LIN {X 0,Y 474.103,Z 226.127,A -85,B 0,C 180,E1 22326.053,E2 22326.053} C_VEL
LIN {X 0,Y 474.112,Z 226.175,A -85,B 0,C 180,E1 22322.417,E2 22322.417} C_VEL
LIN {X 0,Y 474.109,Z 226.126,A -85,B 0,C 180,E1 22318.792,E2 22318.792} C_VEL
LIN {X 0,Y 474.1,Z 226.168,A -85,B 0,C 180,E1 22315.161,E2 22315.161} C_VEL
LIN {X 0,Y 474.084,Z 226.14,A -85,B 0,C 180,E1 22311.559,E2 22311.559} C_VEL
LIN {X 0,Y 474.099,Z 226.178,A -85,B 0,C 180,E1 22307.948,E2 22307.948} C_VEL
LIN {X 0,Y 474.117,Z 226.162,A -85,B 0,C 180,E1 22304.339,E2 22304.339} C_VEL
LIN {X 0,Y 474.116,Z 226.167,A -85,B 0,C 180,E1 22300.664,E2 22300.664} C_VEL
LIN {X 0,Y 474.086,Z 226.178,A -85,B 0,C 180,E1 22297.165,E2 22297.165} C_VEL
LIN {X 0,Y 474.083,Z 226.168,A -85,B 0,C 180,E1 22293.575,E2 22293.575} C_VEL
LIN {X 0,Y 474.134,Z 226.296,A -85,B 0,C 180,E1 22292.55,E2 22292.55} C_VEL
LIN {X 0,Y 475.326,Z 229.528,A -85,B 0,C 180,E1 22292.024,E2 22292.024} C_VEL
LIN {X 0,Y 476.699,Z 231.84,A -85,B 0,C 180,E1 22291.566,E2 22291.566} C_VEL
LIN {X 0,Y 481.647,Z 241.457,A -85,B 0,C 180,E1 22289.842,E2 22289.842} C_VEL
LIN {X 0,Y 489.624,Z 256.766,A -85,B 0,C 180,E1 22287.236,E2 22287.236} C_VEL
LIN {X 0,Y 500.094,Z 277.627,A -85,B 0,C 180,E1 22283.997,E2 22283.997} C_VEL
LIN {X 0,Y 511.483,Z 301.22,A -85,B 0,C 180,E1 22280.7,E2 22280.7} C_VEL
LIN {X 0,Y 519.807,Z 318.56,A -85,B 0,C 180,E1 22278.514,E2 22278.514} C_VEL
LIN {X 0,Y 522.352,Z 322.995,A -85,B 0,C 180,E1 22278.188,E2 22278.188} C_VEL
LIN {X 0,Y 524.642,Z 347.742,A -85,B 0,C 180,E1 22277.464,E2 22277.464} C_VEL
LIN {X 0,Y 513.943,Z 587.488,A -85,B 0,C 180,E1 22273.462,E2 22273.462} C_VEL
LIN {X 0,Y 509.832,Z 692.964,A -85,B 0,C 180,E1 22271.722,E2 22271.722} C_VEL
LIN {X 0,Y 508.032,Z 717.442,A -85,B 0,C 180,E1 22271.132,E2 22271.132} C_VEL
LIN {X 0,Y 505.864,Z 741.406,A -85,B 0,C 180,E1 22270.37,E2 22270.37} C_VEL
LIN {X 0,Y 503.324,Z 764.227,A -85,B 0,C 180,E1 22269.435,E2 22269.435} C_VEL
LIN {X 0,Y 500.285,Z 788.254,A -85,B 0,C 180,E1 22268.236,E2 22268.236} C_VEL
LIN {X 0,Y 497.424,Z 808.594,A -85,B 0,C 180,E1 22267.016,E2 22267.016} C_VEL
LIN {X 0,Y 493.885,Z 831.697,A -85,B 0,C 180,E1 22265.382,E2 22265.382} C_VEL
LIN {X 0,Y 490.913,Z 850.192,A -85,B 0,C 180,E1 22263.853,E2 22263.853} C_VEL
LIN {X 0,Y 487.599,Z 870.092,A -85,B 0,C 180,E1 22261.942,E2 22261.942} C_VEL
LIN {X 0,Y 484.649,Z 887.507,A -85,B 0,C 180,E1 22260.02,E2 22260.02} C_VEL
LIN {X 0,Y 481.773,Z 904.616,A -85,B 0,C 180,E1 22257.838,E2 22257.838} C_VEL
LIN {X 0,Y 479.426,Z 919.191,A -85,B 0,C 180,E1 22255.709,E2 22255.709} C_VEL
LIN {X 0,Y 477.164,Z 934.025,A -85,B 0,C 180,E1 22253.201,E2 22253.201} C_VEL
LIN {X 0,Y 475.501,Z 946.237,A -85,B 0,C 180,E1 22250.816,E2 22250.816} C_VEL
LIN {X 0,Y 474.103,Z 958.209,A -85,B 0,C 180,E1 22248.061,E2 22248.061} C_VEL
LIN {X 0,Y 473.22,Z 967.521,A -85,B 0,C 180,E1 22245.526,E2 22245.526} C_VEL
LIN {X 0,Y 472.64,Z 976.006,A -85,B 0,C 180,E1 22242.71,E2 22242.71} C_VEL
LIN {X 0,Y 472.385,Z 982.114,A -85,B 0,C 180,E1 22240.178,E2 22240.178} C_VEL
LIN {X 0,Y 472.289,Z 987.389,A -85,B 0,C 180,E1 22237.298,E2 22237.298} C_VEL
LIN {X 0,Y 472.333,Z 990.403,A -85,B 0,C 180,E1 22234.857,E2 22234.857} C_VEL
LIN {X 0,Y 472.382,Z 992.129,A -85,B 0,C 180,E1 22232.548,E2 22232.548} C_VEL
LIN {X 0,Y 472.425,Z 992.783,A -85,B 0,C 180,E1 22229.879,E2 22229.879} C_VEL
LIN {X 0,Y 472.4,Z 991.751,A -85,B 0,C 180,E1 22227.21,E2 22227.21} C_VEL
LIN {X 0,Y 472.366,Z 989.7,A -85,B 0,C 180,E1 22224.899,E2 22224.899} C_VEL
LIN {X 0,Y 472.343,Z 986.144,A -85,B 0,C 180,E1 22222.336,E2 22222.336} C_VEL
LIN {X 0,Y 472.457,Z 980.753,A -85,B 0,C 180,E1 22219.636,E2 22219.636} C_VEL
LIN {X 0,Y 472.711,Z 974.464,A -85,B 0,C 180,E1 22217.168,E2 22217.168} C_VEL
LIN {X 0,Y 473.282,Z 965.476,A -85,B 0,C 180,E1 22214.311,E2 22214.311} C_VEL
LIN {X 0,Y 474.142,Z 955.945,A -85,B 0,C 180,E1 22211.814,E2 22211.814} C_VEL
LIN {X 0,Y 475.522,Z 943.625,A -85,B 0,C 180,E1 22209.055,E2 22209.055} C_VEL
LIN {X 0,Y 477.241,Z 930.371,A -85,B 0,C 180,E1 22206.542,E2 22206.542} C_VEL
LIN {X 0,Y 479.545,Z 914.812,A -85,B 0,C 180,E1 22203.984,E2 22203.984} C_VEL
LIN {X 0,Y 482.006,Z 899.256,A -85,B 0,C 180,E1 22201.773,E2 22201.773} C_VEL
LIN {X 0,Y 485.194,Z 880.054,A -85,B 0,C 180,E1 22199.401,E2 22199.401} C_VEL
LIN {X 0,Y 488.36,Z 861.534,A -85,B 0,C 180,E1 22197.42,E2 22197.42} C_VEL
LIN {X 0,Y 491.865,Z 840.855,A -85,B 0,C 180,E1 22195.519,E2 22195.519} C_VEL
LIN {X 0,Y 495.389,Z 819.524,A -85,B 0,C 180,E1 22193.823,E2 22193.823} C_VEL
LIN {X 0,Y 498.74,Z 797.883,A -85,B 0,C 180,E1 22192.365,E2 22192.365} C_VEL
LIN {X 0,Y 502.253,Z 774.045,A -85,B 0,C 180,E1 22191.016,E2 22191.016} C_VEL
LIN {X 0,Y 505.228,Z 751.77,A -85,B 0,C 180,E1 22189.969,E2 22189.969} C_VEL
LIN {X 0,Y 507.919,Z 728.566,A -85,B 0,C 180,E1 22189.093,E2 22189.093} C_VEL
LIN {X 0,Y 510.279,Z 705.051,A -85,B 0,C 180,E1 22188.392,E2 22188.392} C_VEL
LIN {X 0,Y 512.094,Z 679.83,A -85,B 0,C 180,E1 22187.846,E2 22187.846} C_VEL
LIN {X 0,Y 517.017,Z 597.902,A -85,B 0,C 180,E1 22186.328,E2 22186.328} C_VEL
LIN {X 0,Y 522.642,Z 530.22,A -85,B 0,C 180,E1 22184.953,E2 22184.953} C_VEL
LIN {X 0,Y 529.867,Z 464.415,A -85,B 0,C 180,E1 22183.508,E2 22183.508} C_VEL
LIN {X 0,Y 538.765,Z 402.255,A -85,B 0,C 180,E1 22182.087,E2 22182.087} C_VEL
LIN {X 0,Y 544.168,Z 370.237,A -85,B 0,C 180,E1 22181.326,E2 22181.326} C_VEL
LIN {X 0,Y 538.418,Z 386.185,A -85,B 0,C 180,E1 22179.758,E2 22179.758} C_VEL
LIN {X 0,Y 534.921,Z 400.034,A -85,B 0,C 180,E1 22178.53,E2 22178.53} C_VEL
LIN {X 0,Y 531.61,Z 418.651,A -85,B 0,C 180,E1 22177.072,E2 22177.072} C_VEL
LIN {X 0,Y 528.747,Z 441.431,A -85,B 0,C 180,E1 22175.545,E2 22175.545} C_VEL
LIN {X 0,Y 526.309,Z 468.54,A -85,B 0,C 180,E1 22173.972,E2 22173.972} C_VEL
LIN {X 0,Y 524.021,Z 500.146,A -85,B 0,C 180,E1 22172.4,E2 22172.4} C_VEL
LIN {X 0,Y 523.085,Z 512.301,A -85,B 0,C 180,E1 22171.879,E2 22171.879} C_VEL
LIN {X 0,Y 507.968,Z 623.688,A -85,B 0,C 180,E1 22168.838,E2 22168.838} C_VEL
LIN {X 0,Y 500.211,Z 692.312,A -85,B 0,C 180,E1 22166.905,E2 22166.905} C_VEL
LIN {X 0,Y 497.222,Z 717.176,A -85,B 0,C 180,E1 22165.969,E2 22165.969} C_VEL
LIN {X 0,Y 494.515,Z 738.857,A -85,B 0,C 180,E1 22164.934,E2 22164.934} C_VEL
LIN {X 0,Y 491.751,Z 760.438,A -85,B 0,C 180,E1 22163.677,E2 22163.677} C_VEL
LIN {X 0,Y 489.036,Z 780.869,A -85,B 0,C 180,E1 22162.226,E2 22162.226} C_VEL
LIN {X 0,Y 486.605,Z 798.705,A -85,B 0,C 180,E1 22160.697,E2 22160.697} C_VEL
LIN {X 0,Y 484.482,Z 813.948,A -85,B 0,C 180,E1 22159.157,E2 22159.157} C_VEL
LIN {X 0,Y 482.34,Z 828.73,A -85,B 0,C 180,E1 22157.368,E2 22157.368} C_VEL
LIN {X 0,Y 480.502,Z 841.055,A -85,B 0,C 180,E1 22155.572,E2 22155.572} C_VEL
LIN {X 0,Y 478.852,Z 851.963,A -85,B 0,C 180,E1 22153.648,E2 22153.648} C_VEL
LIN {X 0,Y 477.393,Z 861.257,A -85,B 0,C 180,E1 22151.6,E2 22151.6} C_VEL
LIN {X 0,Y 476.233,Z 868.521,A -85,B 0,C 180,E1 22149.548,E2 22149.548} C_VEL
LIN {X 0,Y 475.29,Z 874.171,A -85,B 0,C 180,E1 22147.373,E2 22147.373} C_VEL
LIN {X 0,Y 474.594,Z 877.91,A -85,B 0,C 180,E1 22145.198,E2 22145.198} C_VEL
LIN {X 0,Y 474.097,Z 879.81,A -85,B 0,C 180,E1 22143.022,E2 22143.022} C_VEL
LIN {X 0,Y 473.788,Z 879.972,A -85,B 0,C 180,E1 22140.967,E2 22140.967} C_VEL
LIN {X 0,Y 473.605,Z 878.463,A -85,B 0,C 180,E1 22138.79,E2 22138.79} C_VEL
LIN {X 0,Y 473.549,Z 875.211,A -85,B 0,C 180,E1 22136.611,E2 22136.611} C_VEL
LIN {X 0,Y 473.645,Z 870.182,A -85,B 0,C 180,E1 22134.427,E2 22134.427} C_VEL
LIN {X 0,Y 473.915,Z 863.283,A -85,B 0,C 180,E1 22132.24,E2 22132.24} C_VEL
LIN {X 0,Y 474.405,Z 854.34,A -85,B 0,C 180,E1 22130.048,E2 22130.048} C_VEL
LIN {X 0,Y 475.124,Z 843.798,A -85,B 0,C 180,E1 22127.975,E2 22127.975} C_VEL
LIN {X 0,Y 476.057,Z 831.7,A -85,B 0,C 180,E1 22126.017,E2 22126.017} C_VEL
LIN {X 0,Y 477.184,Z 818.188,A -85,B 0,C 180,E1 22124.193,E2 22124.193} C_VEL
LIN {X 0,Y 478.539,Z 802.58,A -85,B 0,C 180,E1 22122.426,E2 22122.426} C_VEL
LIN {X 0,Y 480.003,Z 785.869,A -85,B 0,C 180,E1 22120.847,E2 22120.847} C_VEL
LIN {X 0,Y 481.552,Z 767.326,A -85,B 0,C 180,E1 22119.393,E2 22119.393} C_VEL
LIN {X 0,Y 483.066,Z 748.687,A -85,B 0,C 180,E1 22118.189,E2 22118.189} C_VEL
LIN {X 0,Y 484.603,Z 728.049,A -85,B 0,C 180,E1 22117.112,E2 22117.112} C_VEL
LIN {X 0,Y 486.002,Z 706.513,A -85,B 0,C 180,E1 22116.236,E2 22116.236} C_VEL
LIN {X 0,Y 487.201,Z 684.993,A -85,B 0,C 180,E1 22115.593,E2 22115.593} C_VEL
LIN {X 0,Y 491.38,Z 580.934,A -85,B 0,C 180,E1 22113.516,E2 22113.516} C_VEL
LIN {X 0,Y 494.767,Z 499.908,A -85,B 0,C 180,E1 22111.921,E2 22111.921} C_VEL
LIN {X 0,Y 489.856,Z 444.398,A -85,B 0,C 180,E1 22110.331,E2 22110.331} C_VEL
LIN {X 0,Y 494.577,Z 391.935,A -85,B 0,C 180,E1 22106.403,E2 22106.403} C_VEL
LIN {X 0,Y 499.626,Z 341.605,A -85,B 0,C 180,E1 22102.609,E2 22102.609} C_VEL
LIN {X 0,Y 504.089,Z 300.496,A -85,B 0,C 180,E1 22099.482,E2 22099.482} C_VEL
LIN {X 0,Y 497.077,Z 281.186,A -85,B 0,C 180,E1 22097.164,E2 22097.164} C_VEL
LIN {X 0,Y 498.864,Z 281.752,A -85,B 0,C 180,E1 22096.884,E2 22096.884} C_VEL
LIN {X 0,Y 503.777,Z 281.964,A -85,B 0,C 180,E1 22096.235,E2 22096.235} C_VEL
LIN {X 0,Y 511.406,Z 300.357,A -85,B 0,C 180,E1 22093.905,E2 22093.905} C_VEL
LIN {X 0,Y 517.83,Z 317.866,A -85,B 0,C 180,E1 22091.832,E2 22091.832} C_VEL
LIN {X 0,Y 517.363,Z 358.606,A -85,B 0,C 180,E1 22089.03,E2 22089.03} C_VEL
LIN {X 0,Y 513.648,Z 376.214,A -85,B 0,C 180,E1 22088.372,E2 22088.372} C_VEL
LIN {X 0,Y 510.519,Z 461.786,A -85,B 0,C 180,E1 22087.05,E2 22087.05} C_VEL
LIN {X 0,Y 507.289,Z 524.733,A -85,B 0,C 180,E1 22085.908,E2 22085.908} C_VEL
LIN {X 0,Y 506.039,Z 532.367,A -85,B 0,C 180,E1 22085.83,E2 22085.83} C_VEL
LIN {X 0,Y 499.793,Z 552.676,A -85,B 0,C 180,E1 22085.852,E2 22085.852} C_VEL
LIN {X 0,Y 498.777,Z 559.214,A -85,B 0,C 180,E1 22085.766,E2 22085.766} C_VEL
LIN {X 0,Y 493.831,Z 632.998,A -85,B 0,C 180,E1 22084.1,E2 22084.1} C_VEL
LIN {X 0,Y 492.338,Z 660.657,A -85,B 0,C 180,E1 22083.328,E2 22083.328} C_VEL
LIN {X 0,Y 490.752,Z 682.372,A -85,B 0,C 180,E1 22082.506,E2 22082.506} C_VEL
LIN {X 0,Y 488.846,Z 702.844,A -85,B 0,C 180,E1 22081.519,E2 22081.519} C_VEL
LIN {X 0,Y 486.522,Z 723.263,A -85,B 0,C 180,E1 22080.301,E2 22080.301} C_VEL
LIN {X 0,Y 483.983,Z 742.53,A -85,B 0,C 180,E1 22078.91,E2 22078.91} C_VEL
LIN {X 0,Y 481.322,Z 760.902,A -85,B 0,C 180,E1 22077.329,E2 22077.329} C_VEL
LIN {X 0,Y 478.596,Z 778.314,A -85,B 0,C 180,E1 22075.558,E2 22075.558} C_VEL
LIN {X 0,Y 476.006,Z 794.203,A -85,B 0,C 180,E1 22073.654,E2 22073.654} C_VEL
LIN {X 0,Y 473.532,Z 809.093,A -85,B 0,C 180,E1 22071.556,E2 22071.556} C_VEL
LIN {X 0,Y 471.329,Z 822.494,A -85,B 0,C 180,E1 22069.326,E2 22069.326} C_VEL
LIN {X 0,Y 469.449,Z 834.427,A -85,B 0,C 180,E1 22066.966,E2 22066.966} C_VEL
LIN {X 0,Y 467.909,Z 844.825,A -85,B 0,C 180,E1 22064.479,E2 22064.479} C_VEL
LIN {X 0,Y 466.793,Z 853.257,A -85,B 0,C 180,E1 22061.992,E2 22061.992} C_VEL
LIN {X 0,Y 466.006,Z 859.958,A -85,B 0,C 180,E1 22059.51,E2 22059.51} C_VEL
LIN {X 0,Y 465.509,Z 865.261,A -85,B 0,C 180,E1 22056.909,E2 22056.909} C_VEL
LIN {X 0,Y 465.23,Z 868.891,A -85,B 0,C 180,E1 22054.314,E2 22054.314} C_VEL
LIN {X 0,Y 465.099,Z 870.797,A -85,B 0,C 180,E1 22051.725,E2 22051.725} C_VEL
LIN {X 0,Y 465.069,Z 871.098,A -85,B 0,C 180,E1 22049.261,E2 22049.261} C_VEL
LIN {X 0,Y 465.149,Z 869.976,A -85,B 0,C 180,E1 22046.796,E2 22046.796} C_VEL
LIN {X 0,Y 465.356,Z 867.167,A -85,B 0,C 180,E1 22044.204,E2 22044.204} C_VEL
LIN {X 0,Y 465.713,Z 862.893,A -85,B 0,C 180,E1 22041.729,E2 22041.729} C_VEL
LIN {X 0,Y 466.373,Z 856.661,A -85,B 0,C 180,E1 22039.096,E2 22039.096} C_VEL
LIN {X 0,Y 467.313,Z 849.17,A -85,B 0,C 180,E1 22036.639,E2 22036.639} C_VEL
LIN {X 0,Y 468.657,Z 839.774,A -85,B 0,C 180,E1 22034.152,E2 22034.152} C_VEL
LIN {X 0,Y 470.425,Z 828.283,A -85,B 0,C 180,E1 22031.665,E2 22031.665} C_VEL
LIN {X 0,Y 472.548,Z 815.17,A -85,B 0,C 180,E1 22029.307,E2 22029.307} C_VEL
LIN {X 0,Y 474.847,Z 801.303,A -85,B 0,C 180,E1 22027.204,E2 22027.204} C_VEL
LIN {X 0,Y 477.37,Z 786.058,A -85,B 0,C 180,E1 22025.234,E2 22025.234} C_VEL
LIN {X 0,Y 480.042,Z 769.347,A -85,B 0,C 180,E1 22023.396,E2 22023.396} C_VEL
LIN {X 0,Y 482.71,Z 751.732,A -85,B 0,C 180,E1 22021.75,E2 22021.75} C_VEL
LIN {X 0,Y 485.282,Z 733.327,A -85,B 0,C 180,E1 22020.295,E2 22020.295} C_VEL
LIN {X 0,Y 487.727,Z 713.336,A -85,B 0,C 180,E1 22018.976,E2 22018.976} C_VEL
LIN {X 0,Y 489.988,Z 691.73,A -85,B 0,C 180,E1 22017.818,E2 22017.818} C_VEL
LIN {X 0,Y 491.801,Z 669.836,A -85,B 0,C 180,E1 22016.893,E2 22016.893} C_VEL
LIN {X 0,Y 493.107,Z 647.709,A -85,B 0,C 180,E1 22016.184,E2 22016.184} C_VEL
LIN {X 0,Y 495.899,Z 602.371,A -85,B 0,C 180,E1 22015.079,E2 22015.079} C_VEL
LIN {X 0,Y 500.552,Z 531.774,A -85,B 0,C 180,E1 22013.579,E2 22013.579} C_VEL
LIN {X 0,Y 504.112,Z 465.945,A -85,B 0,C 180,E1 22012.361,E2 22012.361} C_VEL
LIN {X 0,Y 507.201,Z 385.644,A -85,B 0,C 180,E1 22011.099,E2 22011.099} C_VEL
LIN {X 0,Y 507.596,Z 377.376,A -85,B 0,C 180,E1 22010.96,E2 22010.96} C_VEL
LIN {X 0,Y 511.408,Z 359.689,A -85,B 0,C 180,E1 22010.257,E2 22010.257} C_VEL
LIN {X 0,Y 511.798,Z 321.583,A -85,B 0,C 180,E1 22007.622,E2 22007.622} C_VEL
LIN {X 0,Y 503.702,Z 299.721,A -85,B 0,C 180,E1 22004.967,E2 22004.967} C_VEL
LIN {X 0,Y 495.259,Z 280.206,A -85,B 0,C 180,E1 22002.402,E2 22002.402} C_VEL
LIN {X 0,Y 487.022,Z 263.522,A -85,B 0,C 180,E1 21999.987,E2 21999.987} C_VEL
LIN {X 0,Y 480.126,Z 251.024,A -85,B 0,C 180,E1 21998.057,E2 21998.057} C_VEL
LIN {X 0,Y 474.875,Z 242.046,A -85,B 0,C 180,E1 21996.576,E2 21996.576} C_VEL
LIN {X 0,Y 472.072,Z 237.344,A -85,B 0,C 180,E1 21995.774,E2 21995.774} C_VEL
LIN {X 0,Y 469.994,Z 234.244,A -85,B 0,C 180,E1 21995.208,E2 21995.208} C_VEL
LIN {X 0,Y 469.308,Z 232.581,A -85,B 0,C 180,E1 21994.968,E2 21994.968} C_VEL
LIN {X 0,Y 467.108,Z 230.042,A -85,B 0,C 180,E1 21994.411,E2 21994.411} C_VEL
LIN {X 0,Y 466.171,Z 227.144,A -85,B 0,C 180,E1 21994.006,E2 21994.006} C_VEL
LIN {X 0,Y 466.183,Z 227.157,A -85,B 0,C 180,E1 21990.268,E2 21990.268} C_VEL
LIN {X 0,Y 466.167,Z 227.157,A -85,B 0,C 180,E1 21986.565,E2 21986.565} C_VEL
LIN {X 0,Y 466.163,Z 227.125,A -85,B 0,C 180,E1 21982.845,E2 21982.845} C_VEL
LIN {X 0,Y 466.169,Z 227.13,A -85,B 0,C 180,E1 21979.288,E2 21979.288} C_VEL
LIN {X 0,Y 466.166,Z 227.16,A -85,B 0,C 180,E1 21975.552,E2 21975.552} C_VEL
LIN {X 0,Y 466.157,Z 227.117,A -85,B 0,C 180,E1 21971.883,E2 21971.883} C_VEL
LIN {X 0,Y 466.173,Z 227.152,A -85,B 0,C 180,E1 21968.263,E2 21968.263} C_VEL
LIN {X 0,Y 466.167,Z 227.131,A -85,B 0,C 180,E1 21964.552,E2 21964.552} C_VEL
LIN {X 0,Y 466.172,Z 227.129,A -85,B 0,C 180,E1 21960.86,E2 21960.86} C_VEL
LIN {X 0,Y 466.16,Z 227.153,A -85,B 0,C 180,E1 21957.172,E2 21957.172} C_VEL
LIN {X 0,Y 466.145,Z 227.119,A -85,B 0,C 180,E1 21953.596,E2 21953.596} C_VEL
LIN {X 0,Y 466.16,Z 227.164,A -85,B 0,C 180,E1 21949.91,E2 21949.91} C_VEL
LIN {X 0,Y 466.178,Z 227.164,A -85,B 0,C 180,E1 21946.227,E2 21946.227} C_VEL
LIN {X 0,Y 466.178,Z 227.161,A -85,B 0,C 180,E1 21942.525,E2 21942.525} C_VEL
LIN {X 0,Y 466.164,Z 227.154,A -85,B 0,C 180,E1 21938.878,E2 21938.878} C_VEL
LIN {X 0,Y 466.143,Z 227.158,A -85,B 0,C 180,E1 21935.274,E2 21935.274} C_VEL
LIN {X 0,Y 466.167,Z 227.306,A -85,B 0,C 180,E1 21933.641,E2 21933.641} C_VEL
LIN {X 0,Y 467.547,Z 230.773,A -85,B 0,C 180,E1 21933.039,E2 21933.039} C_VEL
LIN {X 0,Y 468.637,Z 232.398,A -85,B 0,C 180,E1 21932.695,E2 21932.695} C_VEL
LIN {X 0,Y 470.585,Z 236.188,A -85,B 0,C 180,E1 21931.993,E2 21931.993} C_VEL
LIN {X 0,Y 479.969,Z 254.318,A -85,B 0,C 180,E1 21928.753,E2 21928.753} C_VEL
LIN {X 0,Y 490.555,Z 275.349,A -85,B 0,C 180,E1 21925.341,E2 21925.341} C_VEL
LIN {X 0,Y 500.946,Z 296.719,A -85,B 0,C 180,E1 21922.209,E2 21922.209} C_VEL
LIN {X 0,Y 511.695,Z 319.213,A -85,B 0,C 180,E1 21919.239,E2 21919.239} C_VEL
LIN {X 0,Y 516.358,Z 326.875,A -85,B 0,C 180,E1 21918.648,E2 21918.648} C_VEL
LIN {X 0,Y 518.336,Z 348.872,A -85,B 0,C 180,E1 21917.996,E2 21917.996} C_VEL
LIN {X 0,Y 507.238,Z 586.374,A -85,B 0,C 180,E1 21913.964,E2 21913.964} C_VEL
LIN {X 0,Y 502.902,Z 692.911,A -85,B 0,C 180,E1 21912.176,E2 21912.176} C_VEL
LIN {X 0,Y 501.042,Z 717.485,A -85,B 0,C 180,E1 21911.575,E2 21911.575} C_VEL
LIN {X 0,Y 498.81,Z 741.363,A -85,B 0,C 180,E1 21910.805,E2 21910.805} C_VEL
LIN {X 0,Y 496.263,Z 763.656,A -85,B 0,C 180,E1 21909.883,E2 21909.883} C_VEL
LIN {X 0,Y 493.243,Z 787.052,A -85,B 0,C 180,E1 21908.71,E2 21908.71} C_VEL
LIN {X 0,Y 490.284,Z 807.507,A -85,B 0,C 180,E1 21907.475,E2 21907.475} C_VEL
LIN {X 0,Y 486.843,Z 829.512,A -85,B 0,C 180,E1 21905.915,E2 21905.915} C_VEL
LIN {X 0,Y 483.717,Z 848.3,A -85,B 0,C 180,E1 21904.355,E2 21904.355} C_VEL
LIN {X 0,Y 480.169,Z 869.073,A -85,B 0,C 180,E1 21902.355,E2 21902.355} C_VEL
LIN {X 0,Y 477.21,Z 886.031,A -85,B 0,C 180,E1 21900.468,E2 21900.468} C_VEL
LIN {X 0,Y 474.101,Z 903.893,A -85,B 0,C 180,E1 21898.167,E2 21898.167} C_VEL
LIN {X 0,Y 471.568,Z 919.187,A -85,B 0,C 180,E1 21895.899,E2 21895.899} C_VEL
LIN {X 0,Y 469.349,Z 933.266,A -85,B 0,C 180,E1 21893.477,E2 21893.477} C_VEL
LIN {X 0,Y 467.629,Z 945.482,A -85,B 0,C 180,E1 21891.052,E2 21891.052} C_VEL
LIN {X 0,Y 466.173,Z 957.477,A -85,B 0,C 180,E1 21888.249,E2 21888.249} C_VEL
LIN {X 0,Y 465.263,Z 966.781,A -85,B 0,C 180,E1 21885.678,E2 21885.678} C_VEL
LIN {X 0,Y 464.669,Z 975.278,A -85,B 0,C 180,E1 21882.805,E2 21882.805} C_VEL
LIN {X 0,Y 464.416,Z 981.244,A -85,B 0,C 180,E1 21880.286,E2 21880.286} C_VEL
LIN {X 0,Y 464.32,Z 986.433,A -85,B 0,C 180,E1 21877.424,E2 21877.424} C_VEL
LIN {X 0,Y 464.373,Z 989.471,A -85,B 0,C 180,E1 21874.941,E2 21874.941} C_VEL
LIN {X 0,Y 464.429,Z 991.213,A -85,B 0,C 180,E1 21872.591,E2 21872.591} C_VEL
LIN {X 0,Y 464.477,Z 991.875,A -85,B 0,C 180,E1 21869.877,E2 21869.877} C_VEL
LIN {X 0,Y 464.447,Z 990.846,A -85,B 0,C 180,E1 21867.162,E2 21867.162} C_VEL
LIN {X 0,Y 464.405,Z 988.778,A -85,B 0,C 180,E1 21864.812,E2 21864.812} C_VEL
LIN {X 0,Y 464.382,Z 985.207,A -85,B 0,C 180,E1 21862.204,E2 21862.204} C_VEL
LIN {X 0,Y 464.483,Z 979.801,A -85,B 0,C 180,E1 21859.457,E2 21859.457} C_VEL
LIN {X 0,Y 464.771,Z 973.134,A -85,B 0,C 180,E1 21856.818,E2 21856.818} C_VEL
LIN {X 0,Y 465.389,Z 964.01,A -85,B 0,C 180,E1 21853.909,E2 21853.909} C_VEL
LIN {X 0,Y 466.305,Z 954.396,A -85,B 0,C 180,E1 21851.367,E2 21851.367} C_VEL
LIN {X 0,Y 467.802,Z 941.928,A -85,B 0,C 180,E1 21848.562,E2 21848.562} C_VEL
LIN {X 0,Y 469.561,Z 929.295,A -85,B 0,C 180,E1 21846.135,E2 21846.135} C_VEL
LIN {X 0,Y 471.941,Z 914.029,A -85,B 0,C 180,E1 21843.582,E2 21843.582} C_VEL
LIN {X 0,Y 474.607,Z 898.182,A -85,B 0,C 180,E1 21841.292,E2 21841.292} C_VEL
LIN {X 0,Y 477.963,Z 879.004,A -85,B 0,C 180,E1 21838.887,E2 21838.887} C_VEL
LIN {X 0,Y 481.406,Z 860.028,A -85,B 0,C 180,E1 21836.829,E2 21836.829} C_VEL
LIN {X 0,Y 485.017,Z 839.842,A -85,B 0,C 180,E1 21834.953,E2 21834.953} C_VEL
LIN {X 0,Y 488.706,Z 818.705,A -85,B 0,C 180,E1 21833.247,E2 21833.247} C_VEL
LIN {X 0,Y 492.221,Z 797.381,A -85,B 0,C 180,E1 21831.789,E2 21831.789} C_VEL
LIN {X 0,Y 495.94,Z 773.646,A -85,B 0,C 180,E1 21830.424,E2 21830.424} C_VEL
LIN {X 0,Y 499.069,Z 751.686,A -85,B 0,C 180,E1 21829.372,E2 21829.372} C_VEL
LIN {X 0,Y 501.964,Z 728.472,A -85,B 0,C 180,E1 21828.477,E2 21828.477} C_VEL
LIN {X 0,Y 504.399,Z 706.193,A -85,B 0,C 180,E1 21827.792,E2 21827.792} C_VEL
LIN {X 0,Y 506.382,Z 681.601,A -85,B 0,C 180,E1 21827.233,E2 21827.233} C_VEL
LIN {X 0,Y 511.96,Z 599.732,A -85,B 0,C 180,E1 21825.657,E2 21825.657} C_VEL
LIN {X 0,Y 518.163,Z 533.367,A -85,B 0,C 180,E1 21824.262,E2 21824.262} C_VEL
LIN {X 0,Y 525.811,Z 470.913,A -85,B 0,C 180,E1 21822.85,E2 21822.85} C_VEL
LIN {X 0,Y 535.086,Z 411.727,A -85,B 0,C 180,E1 21821.472,E2 21821.472} C_VEL
LIN {X 0,Y 539.64,Z 386.423,A -85,B 0,C 180,E1 21820.867,E2 21820.867} C_VEL
LIN {X 0,Y 534.431,Z 402.446,A -85,B 0,C 180,E1 21819.41,E2 21819.41} C_VEL
LIN {X 0,Y 530.546,Z 419.16,A -85,B 0,C 180,E1 21818.062,E2 21818.062} C_VEL
LIN {X 0,Y 526.896,Z 440.675,A -85,B 0,C 180,E1 21816.55,E2 21816.55} C_VEL
LIN {X 0,Y 523.592,Z 467.503,A -85,B 0,C 180,E1 21814.928,E2 21814.928} C_VEL
LIN {X 0,Y 520.576,Z 498.689,A -85,B 0,C 180,E1 21813.313,E2 21813.313} C_VEL
LIN {X 0,Y 519.163,Z 513.949,A -85,B 0,C 180,E1 21812.626,E2 21812.626} C_VEL
LIN {X 0,Y 503.179,Z 623.523,A -85,B 0,C 180,E1 21809.575,E2 21809.575} C_VEL
LIN {X 0,Y 494.715,Z 692.559,A -85,B 0,C 180,E1 21807.579,E2 21807.579} C_VEL
LIN {X 0,Y 491.531,Z 716.722,A -85,B 0,C 180,E1 21806.651,E2 21806.651} C_VEL
LIN {X 0,Y 488.391,Z 739.771,A -85,B 0,C 180,E1 21805.529,E2 21805.529} C_VEL
LIN {X 0,Y 485.547,Z 760.078,A -85,B 0,C 180,E1 21804.322,E2 21804.322} C_VEL
LIN {X 0,Y 482.62,Z 780.56,A -85,B 0,C 180,E1 21802.859,E2 21802.859} C_VEL
LIN {X 0,Y 479.706,Z 800.352,A -85,B 0,C 180,E1 21801.137,E2 21801.137} C_VEL
LIN {X 0,Y 477.171,Z 816.917,A -85,B 0,C 180,E1 21799.398,E2 21799.398} C_VEL
LIN {X 0,Y 475.127,Z 830.018,A -85,B 0,C 180,E1 21797.767,E2 21797.767} C_VEL
LIN {X 0,Y 473.167,Z 842.333,A -85,B 0,C 180,E1 21795.945,E2 21795.945} C_VEL
LIN {X 0,Y 471.382,Z 853.157,A -85,B 0,C 180,E1 21793.994,E2 21793.994} C_VEL
LIN {X 0,Y 469.813,Z 862.453,A -85,B 0,C 180,E1 21791.914,E2 21791.914} C_VEL
LIN {X 0,Y 468.488,Z 870.052,A -85,B 0,C 180,E1 21789.707,E2 21789.707} C_VEL
LIN {X 0,Y 467.481,Z 875.602,A -85,B 0,C 180,E1 21787.497,E2 21787.497} C_VEL
LIN {X 0,Y 466.732,Z 879.228,A -85,B 0,C 180,E1 21785.286,E2 21785.286} C_VEL
LIN {X 0,Y 466.2,Z 881.03,A -85,B 0,C 180,E1 21783.074,E2 21783.074} C_VEL
LIN {X 0,Y 465.854,Z 881.048,A -85,B 0,C 180,E1 21780.861,E2 21780.861} C_VEL
LIN {X 0,Y 465.66,Z 879.31,A -85,B 0,C 180,E1 21778.647,E2 21778.647} C_VEL
LIN {X 0,Y 465.608,Z 875.845,A -85,B 0,C 180,E1 21776.429,E2 21776.429} C_VEL
LIN {X 0,Y 465.719,Z 870.596,A -85,B 0,C 180,E1 21774.208,E2 21774.208} C_VEL
LIN {X 0,Y 466.015,Z 863.458,A -85,B 0,C 180,E1 21771.983,E2 21771.983} C_VEL
LIN {X 0,Y 466.507,Z 854.813,A -85,B 0,C 180,E1 21769.877,E2 21769.877} C_VEL
LIN {X 0,Y 467.208,Z 844.805,A -85,B 0,C 180,E1 21767.893,E2 21767.893} C_VEL
LIN {X 0,Y 468.166,Z 832.719,A -85,B 0,C 180,E1 21765.908,E2 21765.908} C_VEL
LIN {X 0,Y 469.327,Z 819.151,A -85,B 0,C 180,E1 21764.048,E2 21764.048} C_VEL
LIN {X 0,Y 470.666,Z 804.108,A -85,B 0,C 180,E1 21762.314,E2 21762.314} C_VEL
LIN {X 0,Y 472.163,Z 787.528,A -85,B 0,C 180,E1 21760.709,E2 21760.709} C_VEL
LIN {X 0,Y 473.767,Z 769.076,A -85,B 0,C 180,E1 21759.221,E2 21759.221} C_VEL
LIN {X 0,Y 475.377,Z 749.813,A -85,B 0,C 180,E1 21757.948,E2 21757.948} C_VEL
LIN {X 0,Y 476.956,Z 729.338,A -85,B 0,C 180,E1 21756.854,E2 21756.854} C_VEL
LIN {X 0,Y 478.443,Z 707.237,A -85,B 0,C 180,E1 21755.934,E2 21755.934} C_VEL
LIN {X 0,Y 479.691,Z 685.63,A -85,B 0,C 180,E1 21755.271,E2 21755.271} C_VEL
LIN {X 0,Y 481.691,Z 636.241,A -85,B 0,C 180,E1 21754.247,E2 21754.247} C_VEL
LIN {X 0,Y 487.592,Z 500.852,A -85,B 0,C 180,E1 21751.518,E2 21751.518} C_VEL
LIN {X 0,Y 482.649,Z 443.526,A -85,B 0,C 180,E1 21749.842,E2 21749.842} C_VEL
LIN {X 0,Y 487.555,Z 391.321,A -85,B 0,C 180,E1 21745.886,E2 21745.886} C_VEL
LIN {X 0,Y 492.883,Z 340.388,A -85,B 0,C 180,E1 21741.997,E2 21741.997} C_VEL
LIN {X 0,Y 497.018,Z 303.388,A -85,B 0,C 180,E1 21739.151,E2 21739.151} C_VEL
LIN {X 0,Y 491.675,Z 288.4,A -85,B 0,C 180,E1 21737.335,E2 21737.335} C_VEL
LIN {X 0,Y 493.95,Z 288.989,A -85,B 0,C 180,E1 21736.985,E2 21736.985} C_VEL
LIN {X 0,Y 499.293,Z 289.309,A -85,B 0,C 180,E1 21736.259,E2 21736.259} C_VEL
LIN {X 0,Y 507.081,Z 308.783,A -85,B 0,C 180,E1 21733.798,E2 21733.798} C_VEL
LIN {X 0,Y 511.777,Z 322.105,A -85,B 0,C 180,E1 21732.228,E2 21732.228} C_VEL
LIN {X 0,Y 511.313,Z 360.22,A -85,B 0,C 180,E1 21729.602,E2 21729.602} C_VEL
LIN {X 0,Y 507.373,Z 378.886,A -85,B 0,C 180,E1 21728.904,E2 21728.904} C_VEL
LIN {X 0,Y 504.154,Z 463.908,A -85,B 0,C 180,E1 21727.578,E2 21727.578} C_VEL
LIN {X 0,Y 500.507,Z 531.887,A -85,B 0,C 180,E1 21726.323,E2 21726.323} C_VEL
LIN {X 0,Y 498.777,Z 559.214,A -85,B 0,C 180,E1 21725.766,E2 21725.766} C_VEL
LIN {X 0,Y 497.486,Z 566.831,A -85,B 0,C 180,E1 21725.674,E2 21725.674} C_VEL
LIN {X 0,Y 491.089,Z 587.097,A -85,B 0,C 180,E1 21725.67,E2 21725.67} C_VEL
LIN {X 0,Y 490.025,Z 593.617,A -85,B 0,C 180,E1 21725.574,E2 21725.574} C_VEL
LIN {X 0,Y 486.575,Z 645.419,A -85,B 0,C 180,E1 21724.314,E2 21724.314} C_VEL
LIN {X 0,Y 485.245,Z 667.881,A -85,B 0,C 180,E1 21723.614,E2 21723.614} C_VEL
LIN {X 0,Y 483.547,Z 688.635,A -85,B 0,C 180,E1 21722.761,E2 21722.761} C_VEL
LIN {X 0,Y 481.427,Z 709.184,A -85,B 0,C 180,E1 21721.7,E2 21721.7} C_VEL
LIN {X 0,Y 478.958,Z 729.358,A -85,B 0,C 180,E1 21720.422,E2 21720.422} C_VEL
LIN {X 0,Y 476.375,Z 747.976,A -85,B 0,C 180,E1 21719.003,E2 21719.003} C_VEL
LIN {X 0,Y 473.544,Z 766.359,A -85,B 0,C 180,E1 21717.339,E2 21717.339} C_VEL
LIN {X 0,Y 470.669,Z 783.837,A -85,B 0,C 180,E1 21715.461,E2 21715.461} C_VEL
LIN {X 0,Y 467.905,Z 799.872,A -85,B 0,C 180,E1 21713.42,E2 21713.42} C_VEL
LIN {X 0,Y 465.271,Z 814.963,A -85,B 0,C 180,E1 21711.142,E2 21711.142} C_VEL
LIN {X 0,Y 463.008,Z 828.125,A -85,B 0,C 180,E1 21708.77,E2 21708.77} C_VEL
LIN {X 0,Y 461.172,Z 839.251,A -85,B 0,C 180,E1 21706.371,E2 21706.371} C_VEL
LIN {X 0,Y 459.702,Z 848.945,A -85,B 0,C 180,E1 21703.843,E2 21703.843} C_VEL
LIN {X 0,Y 458.578,Z 857.298,A -85,B 0,C 180,E1 21701.13,E2 21701.13} C_VEL
LIN {X 0,Y 457.875,Z 863.459,A -85,B 0,C 180,E1 21698.54,E2 21698.54} C_VEL
LIN {X 0,Y 457.457,Z 868.051,A -85,B 0,C 180,E1 21695.897,E2 21695.897} C_VEL
LIN {X 0,Y 457.224,Z 870.89,A -85,B 0,C 180,E1 21693.26,E2 21693.26} C_VEL
LIN {X 0,Y 457.135,Z 872.082,A -85,B 0,C 180,E1 21690.752,E2 21690.752} C_VEL
LIN {X 0,Y 457.162,Z 871.849,A -85,B 0,C 180,E1 21688.245,E2 21688.245} C_VEL
LIN {X 0,Y 457.302,Z 869.964,A -85,B 0,C 180,E1 21685.597,E2 21685.597} C_VEL
LIN {X 0,Y 457.597,Z 866.416,A -85,B 0,C 180,E1 21682.971,E2 21682.971} C_VEL
LIN {X 0,Y 458.118,Z 861.185,A -85,B 0,C 180,E1 21680.325,E2 21680.325} C_VEL
LIN {X 0,Y 458.958,Z 854.552,A -85,B 0,C 180,E1 21677.8,E2 21677.8} C_VEL
LIN {X 0,Y 460.152,Z 846.045,A -85,B 0,C 180,E1 21675.233,E2 21675.233} C_VEL
LIN {X 0,Y 461.846,Z 835.297,A -85,B 0,C 180,E1 21672.616,E2 21672.616} C_VEL
LIN {X 0,Y 463.962,Z 822.671,A -85,B 0,C 180,E1 21670.092,E2 21670.092} C_VEL
LIN {X 0,Y 466.31,Z 809.091,A -85,B 0,C 180,E1 21667.828,E2 21667.828} C_VEL
LIN {X 0,Y 468.767,Z 794.94,A -85,B 0,C 180,E1 21665.824,E2 21665.824} C_VEL
LIN {X 0,Y 471.488,Z 778.982,A -85,B 0,C 180,E1 21663.893,E2 21663.893} C_VEL
LIN {X 0,Y 474.336,Z 761.484,A -85,B 0,C 180,E1 21662.097,E2 21662.097} C_VEL
LIN {X 0,Y 477.008,Z 743.797,A -85,B 0,C 180,E1 21660.557,E2 21660.557} C_VEL
LIN {X 0,Y 479.644,Z 724.54,A -85,B 0,C 180,E1 21659.148,E2 21659.148} C_VEL
LIN {X 0,Y 482.044,Z 704.365,A -85,B 0,C 180,E1 21657.926,E2 21657.926} C_VEL
LIN {X 0,Y 484.165,Z 682.397,A -85,B 0,C 180,E1 21656.855,E2 21656.855} C_VEL
LIN {X 0,Y 485.877,Z 659.344,A -85,B 0,C 180,E1 21655.992,E2 21655.992} C_VEL
LIN {X 0,Y 487.914,Z 623.727,A -85,B 0,C 180,E1 21655.033,E2 21655.033} C_VEL
LIN {X 0,Y 492.911,Z 552.333,A -85,B 0,C 180,E1 21653.43,E2 21653.43} C_VEL
LIN {X 0,Y 496.796,Z 487.533,A -85,B 0,C 180,E1 21652.165,E2 21652.165} C_VEL
LIN {X 0,Y 499.705,Z 423.65,A -85,B 0,C 180,E1 21651.096,E2 21651.096} C_VEL
LIN {X 0,Y 501.36,Z 380.151,A -85,B 0,C 180,E1 21650.417,E2 21650.417} C_VEL
LIN {X 0,Y 505.415,Z 361.597,A -85,B 0,C 180,E1 21649.69,E2 21649.69} C_VEL
LIN {X 0,Y 505.768,Z 325.409,A -85,B 0,C 180,E1 21647.177,E2 21647.177} C_VEL
LIN {X 0,Y 497.877,Z 304.182,A -85,B 0,C 180,E1 21644.58,E2 21644.58} C_VEL
LIN {X 0,Y 489.767,Z 285.201,A -85,B 0,C 180,E1 21642.039,E2 21642.039} C_VEL
LIN {X 0,Y 481.64,Z 268.543,A -85,B 0,C 180,E1 21639.594,E2 21639.594} C_VEL
LIN {X 0,Y 474.838,Z 256.177,A -85,B 0,C 180,E1 21637.638,E2 21637.638} C_VEL
LIN {X 0,Y 470.082,Z 247.938,A -85,B 0,C 180,E1 21636.251,E2 21636.251} C_VEL
LIN {X 0,Y 467.272,Z 243.314,A -85,B 0,C 180,E1 21635.444,E2 21635.444} C_VEL
LIN {X 0,Y 464.53,Z 238.712,A -85,B 0,C 180,E1 21634.629,E2 21634.629} C_VEL
LIN {X 0,Y 462.104,Z 235.133,A -85,B 0,C 180,E1 21633.935,E2 21633.935} C_VEL
LIN {X 0,Y 461.413,Z 233.57,A -85,B 0,C 180,E1 21633.694,E2 21633.694} C_VEL
LIN {X 0,Y 459.273,Z 231.197,A -85,B 0,C 180,E1 21633.124,E2 21633.124} C_VEL
LIN {X 0,Y 458.221,Z 228.122,A -85,B 0,C 180,E1 21632.689,E2 21632.689} C_VEL
LIN {X 0,Y 458.227,Z 228.119,A -85,B 0,C 180,E1 21628.953,E2 21628.953} C_VEL
LIN {X 0,Y 458.232,Z 228.139,A -85,B 0,C 180,E1 21625.321,E2 21625.321} C_VEL
LIN {X 0,Y 458.229,Z 228.136,A -85,B 0,C 180,E1 21621.633,E2 21621.633} C_VEL
LIN {X 0,Y 458.225,Z 228.105,A -85,B 0,C 180,E1 21617.919,E2 21617.919} C_VEL
LIN {X 0,Y 458.235,Z 228.133,A -85,B 0,C 180,E1 21614.146,E2 21614.146} C_VEL
LIN {X 0,Y 458.231,Z 228.13,A -85,B 0,C 180,E1 21610.435,E2 21610.435} C_VEL
LIN {X 0,Y 458.23,Z 228.107,A -85,B 0,C 180,E1 21606.767,E2 21606.767} C_VEL
LIN {X 0,Y 458.23,Z 228.15,A -85,B 0,C 180,E1 21603.002,E2 21603.002} C_VEL
LIN {X 0,Y 458.214,Z 228.1,A -85,B 0,C 180,E1 21599.375,E2 21599.375} C_VEL
LIN {X 0,Y 458.213,Z 228.15,A -85,B 0,C 180,E1 21595.62,E2 21595.62} C_VEL
LIN {X 0,Y 458.218,Z 228.106,A -85,B 0,C 180,E1 21591.972,E2 21591.972} C_VEL
LIN {X 0,Y 458.234,Z 228.151,A -85,B 0,C 180,E1 21588.292,E2 21588.292} C_VEL
LIN {X 0,Y 458.242,Z 228.138,A -85,B 0,C 180,E1 21584.561,E2 21584.561} C_VEL
LIN {X 0,Y 458.227,Z 228.143,A -85,B 0,C 180,E1 21580.882,E2 21580.882} C_VEL
LIN {X 0,Y 458.206,Z 228.157,A -85,B 0,C 180,E1 21577.279,E2 21577.279} C_VEL
LIN {X 0,Y 458.248,Z 228.309,A -85,B 0,C 180,E1 21574.784,E2 21574.784} C_VEL
LIN {X 0,Y 459.502,Z 231.574,A -85,B 0,C 180,E1 21574.201,E2 21574.201} C_VEL
LIN {X 0,Y 460.611,Z 233.05,A -85,B 0,C 180,E1 21573.853,E2 21573.853} C_VEL
LIN {X 0,Y 462.422,Z 236.877,A -85,B 0,C 180,E1 21573.133,E2 21573.133} C_VEL
LIN {X 0,Y 470.046,Z 251.38,A -85,B 0,C 180,E1 21570.428,E2 21570.428} C_VEL
LIN {X 0,Y 479.662,Z 270.434,A -85,B 0,C 180,E1 21567.181,E2 21567.181} C_VEL
LIN {X 0,Y 489.067,Z 289.421,A -85,B 0,C 180,E1 21564.216,E2 21564.216} C_VEL
LIN {X 0,Y 499.32,Z 310.731,A -85,B 0,C 180,E1 21561.187,E2 21561.187} C_VEL
LIN {X 0,Y 504.05,Z 320.505,A -85,B 0,C 180,E1 21559.93,E2 21559.93} C_VEL
LIN {X 0,Y 510.322,Z 330.764,A -85,B 0,C 180,E1 21559.106,E2 21559.106} C_VEL
LIN {X 0,Y 511.985,Z 350.164,A -85,B 0,C 180,E1 21558.526,E2 21558.526} C_VEL
LIN {X 0,Y 500.204,Z 594.045,A -85,B 0,C 180,E1 21554.333,E2 21554.333} C_VEL
LIN {X 0,Y 495.978,Z 693.246,A -85,B 0,C 180,E1 21552.634,E2 21552.634} C_VEL
LIN {X 0,Y 494.054,Z 717.678,A -85,B 0,C 180,E1 21552.024,E2 21552.024} C_VEL
LIN {X 0,Y 491.76,Z 741.384,A -85,B 0,C 180,E1 21551.246,E2 21551.246} C_VEL
LIN {X 0,Y 489.157,Z 763.478,A -85,B 0,C 180,E1 21550.319,E2 21550.319} C_VEL
LIN {X 0,Y 486.107,Z 786.461,A -85,B 0,C 180,E1 21549.153,E2 21549.153} C_VEL
LIN {X 0,Y 482.946,Z 807.676,A -85,B 0,C 180,E1 21547.854,E2 21547.854} C_VEL
LIN {X 0,Y 479.236,Z 830.66,A -85,B 0,C 180,E1 21546.19,E2 21546.19} C_VEL
LIN {X 0,Y 475.951,Z 849.917,A -85,B 0,C 180,E1 21544.557,E2 21544.557} C_VEL
LIN {X 0,Y 472.486,Z 869.477,A -85,B 0,C 180,E1 21542.62,E2 21542.62} C_VEL
LIN {X 0,Y 469.3,Z 887.249,A -85,B 0,C 180,E1 21540.597,E2 21540.597} C_VEL
LIN {X 0,Y 466.342,Z 903.708,A -85,B 0,C 180,E1 21538.424,E2 21538.424} C_VEL
LIN {X 0,Y 463.846,Z 918.314,A -85,B 0,C 180,E1 21536.226,E2 21536.226} C_VEL
LIN {X 0,Y 461.437,Z 933.109,A -85,B 0,C 180,E1 21533.633,E2 21533.633} C_VEL
LIN {X 0,Y 459.594,Z 945.92,A -85,B 0,C 180,E1 21531.037,E2 21531.037} C_VEL
LIN {X 0,Y 458.192,Z 957.214,A -85,B 0,C 180,E1 21528.315,E2 21528.315} C_VEL
LIN {X 0,Y 457.245,Z 966.776,A -85,B 0,C 180,E1 21525.603,E2 21525.603} C_VEL
LIN {X 0,Y 456.681,Z 974.841,A -85,B 0,C 180,E1 21522.776,E2 21522.776} C_VEL
LIN {X 0,Y 456.438,Z 980.733,A -85,B 0,C 180,E1 21520.221,E2 21520.221} C_VEL
LIN {X 0,Y 456.363,Z 985.805,A -85,B 0,C 180,E1 21517.301,E2 21517.301} C_VEL
LIN {X 0,Y 456.421,Z 988.645,A -85,B 0,C 180,E1 21514.901,E2 21514.901} C_VEL
LIN {X 0,Y 456.484,Z 990.35,A -85,B 0,C 180,E1 21512.511,E2 21512.511} C_VEL
LIN {X 0,Y 456.52,Z 990.948,A -85,B 0,C 180,E1 21509.749,E2 21509.749} C_VEL
LIN {X 0,Y 456.496,Z 989.935,A -85,B 0,C 180,E1 21507.112,E2 21507.112} C_VEL
LIN {X 0,Y 456.445,Z 987.861,A -85,B 0,C 180,E1 21504.721,E2 21504.721} C_VEL
LIN {X 0,Y 456.426,Z 984.128,A -85,B 0,C 180,E1 21501.972,E2 21501.972} C_VEL
LIN {X 0,Y 456.512,Z 978.559,A -85,B 0,C 180,E1 21499.143,E2 21499.143} C_VEL
LIN {X 0,Y 456.806,Z 972.154,A -85,B 0,C 180,E1 21496.584,E2 21496.584} C_VEL
LIN {X 0,Y 457.471,Z 963.024,A -85,B 0,C 180,E1 21493.623,E2 21493.623} C_VEL
LIN {X 0,Y 458.432,Z 953.388,A -85,B 0,C 180,E1 21491.035,E2 21491.035} C_VEL
LIN {X 0,Y 460.047,Z 940.686,A -85,B 0,C 180,E1 21488.136,E2 21488.136} C_VEL
LIN {X 0,Y 461.929,Z 928.114,A -85,B 0,C 180,E1 21485.686,E2 21485.686} C_VEL
LIN {X 0,Y 464.561,Z 912.168,A -85,B 0,C 180,E1 21482.99,E2 21482.99} C_VEL
LIN {X 0,Y 467.24,Z 897.186,A -85,B 0,C 180,E1 21480.796,E2 21480.796} C_VEL
LIN {X 0,Y 470.791,Z 878.062,A -85,B 0,C 180,E1 21478.359,E2 21478.359} C_VEL
LIN {X 0,Y 474.441,Z 859.063,A -85,B 0,C 180,E1 21476.266,E2 21476.266} C_VEL
LIN {X 0,Y 478.199,Z 839.149,A -85,B 0,C 180,E1 21474.385,E2 21474.385} C_VEL
LIN {X 0,Y 482.12,Z 818.027,A -85,B 0,C 180,E1 21472.654,E2 21472.654} C_VEL
LIN {X 0,Y 485.785,Z 797.142,A -85,B 0,C 180,E1 21471.202,E2 21471.202} C_VEL
LIN {X 0,Y 489.724,Z 773.628,A -85,B 0,C 180,E1 21469.82,E2 21469.82} C_VEL
LIN {X 0,Y 493.009,Z 752.05,A -85,B 0,C 180,E1 21468.765,E2 21468.765} C_VEL
LIN {X 0,Y 496.262,Z 727.875,A -85,B 0,C 180,E1 21467.811,E2 21467.811} C_VEL
LIN {X 0,Y 498.951,Z 704.878,A -85,B 0,C 180,E1 21467.094,E2 21467.094} C_VEL
LIN {X 0,Y 501.206,Z 679.012,A -85,B 0,C 180,E1 21466.502,E2 21466.502} C_VEL
LIN {X 0,Y 506.91,Z 604.456,A -85,B 0,C 180,E1 21465.016,E2 21465.016} C_VEL
LIN {X 0,Y 513.515,Z 540.682,A -85,B 0,C 180,E1 21463.636,E2 21463.636} C_VEL
LIN {X 0,Y 521.895,Z 478.411,A -85,B 0,C 180,E1 21462.196,E2 21462.196} C_VEL
LIN {X 0,Y 532.261,Z 418.01,A -85,B 0,C 180,E1 21460.768,E2 21460.768} C_VEL
LIN {X 0,Y 535.068,Z 403.51,A -85,B 0,C 180,E1 21460.407,E2 21460.407} C_VEL
LIN {X 0,Y 529.965,Z 420.849,A -85,B 0,C 180,E1 21458.976,E2 21458.976} C_VEL
LIN {X 0,Y 525.36,Z 442.234,A -85,B 0,C 180,E1 21457.44,E2 21457.44} C_VEL
LIN {X 0,Y 521.359,Z 467.462,A -85,B 0,C 180,E1 21455.867,E2 21455.867} C_VEL
LIN {X 0,Y 517.712,Z 496.915,A -85,B 0,C 180,E1 21454.28,E2 21454.28} C_VEL
LIN {X 0,Y 515.606,Z 515.721,A -85,B 0,C 180,E1 21453.398,E2 21453.398} C_VEL
LIN {X 0,Y 498.716,Z 623.519,A -85,B 0,C 180,E1 21450.343,E2 21450.343} C_VEL
LIN {X 0,Y 489.462,Z 693.045,A -85,B 0,C 180,E1 21448.282,E2 21448.282} C_VEL
LIN {X 0,Y 485.921,Z 717.566,A -85,B 0,C 180,E1 21447.314,E2 21447.314} C_VEL
LIN {X 0,Y 482.406,Z 741.177,A -85,B 0,C 180,E1 21446.133,E2 21446.133} C_VEL
LIN {X 0,Y 479.01,Z 763.375,A -85,B 0,C 180,E1 21444.766,E2 21444.766} C_VEL
LIN {X 0,Y 475.96,Z 782.652,A -85,B 0,C 180,E1 21443.328,E2 21443.328} C_VEL
LIN {X 0,Y 473.172,Z 800.284,A -85,B 0,C 180,E1 21441.769,E2 21441.769} C_VEL
LIN {X 0,Y 470.431,Z 816.956,A -85,B 0,C 180,E1 21440.011,E2 21440.011} C_VEL
LIN {X 0,Y 467.973,Z 831.456,A -85,B 0,C 180,E1 21438.177,E2 21438.177} C_VEL
LIN {X 0,Y 465.858,Z 843.626,A -85,B 0,C 180,E1 21436.33,E2 21436.33} C_VEL
LIN {X 0,Y 463.953,Z 854.446,A -85,B 0,C 180,E1 21434.35,E2 21434.35} C_VEL
LIN {X 0,Y 462.258,Z 863.686,A -85,B 0,C 180,E1 21432.238,E2 21432.238} C_VEL
LIN {X 0,Y 460.893,Z 870.899,A -85,B 0,C 180,E1 21430.121,E2 21430.121} C_VEL
LIN {X 0,Y 459.777,Z 876.529,A -85,B 0,C 180,E1 21427.875,E2 21427.875} C_VEL
LIN {X 0,Y 458.985,Z 880.06,A -85,B 0,C 180,E1 21425.751,E2 21425.751} C_VEL
LIN {X 0,Y 458.376,Z 882.037,A -85,B 0,C 180,E1 21423.502,E2 21423.502} C_VEL
LIN {X 0,Y 457.98,Z 882.254,A -85,B 0,C 180,E1 21421.251,E2 21421.251} C_VEL
LIN {X 0,Y 457.742,Z 880.699,A -85,B 0,C 180,E1 21418.999,E2 21418.999} C_VEL
LIN {X 0,Y 457.661,Z 877.402,A -85,B 0,C 180,E1 21416.744,E2 21416.744} C_VEL
LIN {X 0,Y 457.746,Z 872.332,A -85,B 0,C 180,E1 21414.485,E2 21414.485} C_VEL
LIN {X 0,Y 458.022,Z 865.378,A -85,B 0,C 180,E1 21412.221,E2 21412.221} C_VEL
LIN {X 0,Y 458.534,Z 856.372,A -85,B 0,C 180,E1 21409.953,E2 21409.953} C_VEL
LIN {X 0,Y 459.29,Z 845.771,A -85,B 0,C 180,E1 21407.809,E2 21407.809} C_VEL
LIN {X 0,Y 460.275,Z 833.663,A -85,B 0,C 180,E1 21405.79,E2 21405.79} C_VEL
LIN {X 0,Y 461.471,Z 820.087,A -85,B 0,C 180,E1 21403.898,E2 21403.898} C_VEL
LIN {X 0,Y 462.908,Z 804.481,A -85,B 0,C 180,E1 21402.073,E2 21402.073} C_VEL
LIN {X 0,Y 464.458,Z 787.813,A -85,B 0,C 180,E1 21400.442,E2 21400.442} C_VEL
LIN {X 0,Y 466.117,Z 769.248,A -85,B 0,C 180,E1 21398.93,E2 21398.93} C_VEL
LIN {X 0,Y 467.783,Z 749.889,A -85,B 0,C 180,E1 21397.637,E2 21397.637} C_VEL
LIN {X 0,Y 469.412,Z 729.333,A -85,B 0,C 180,E1 21396.526,E2 21396.526} C_VEL
LIN {X 0,Y 470.946,Z 707.195,A -85,B 0,C 180,E1 21395.593,E2 21395.593} C_VEL
LIN {X 0,Y 472.25,Z 685.306,A -85,B 0,C 180,E1 21394.913,E2 21394.913} C_VEL
LIN {X 0,Y 476.139,Z 594.578,A -85,B 0,C 180,E1 21393.022,E2 21393.022} C_VEL
LIN {X 0,Y 480.399,Z 501.63,A -85,B 0,C 180,E1 21391.107,E2 21391.107} C_VEL
LIN {X 0,Y 475.428,Z 442.959,A -85,B 0,C 180,E1 21389.367,E2 21389.367} C_VEL
LIN {X 0,Y 480.616,Z 390.245,A -85,B 0,C 180,E1 21385.319,E2 21385.319} C_VEL
LIN {X 0,Y 486.158,Z 339.219,A -85,B 0,C 180,E1 21381.375,E2 21381.375} C_VEL
LIN {X 0,Y 489.964,Z 306.282,A -85,B 0,C 180,E1 21378.81,E2 21378.81} C_VEL
LIN {X 0,Y 486.224,Z 295.751,A -85,B 0,C 180,E1 21377.512,E2 21377.512} C_VEL
LIN {X 0,Y 488.357,Z 296.309,A -85,B 0,C 180,E1 21377.175,E2 21377.175} C_VEL
LIN {X 0,Y 494.683,Z 296.459,A -85,B 0,C 180,E1 21376.309,E2 21376.309} C_VEL
LIN {X 0,Y 502.56,Z 316.624,A -85,B 0,C 180,E1 21373.761,E2 21373.761} C_VEL
LIN {X 0,Y 505.822,Z 326.064,A -85,B 0,C 180,E1 21372.662,E2 21372.662} C_VEL
LIN {X 0,Y 505.293,Z 362.094,A -85,B 0,C 180,E1 21370.173,E2 21370.173} C_VEL
LIN {X 0,Y 501.139,Z 381.657,A -85,B 0,C 180,E1 21369.448,E2 21369.448} C_VEL
LIN {X 0,Y 497.822,Z 466.245,A -85,B 0,C 180,E1 21368.115,E2 21368.115} C_VEL
LIN {X 0,Y 494.1,Z 533.338,A -85,B 0,C 180,E1 21366.862,E2 21366.862} C_VEL
LIN {X 0,Y 490.025,Z 593.617,A -85,B 0,C 180,E1 21365.574,E2 21365.574} C_VEL
LIN {X 0,Y 488.675,Z 601.21,A -85,B 0,C 180,E1 21365.469,E2 21365.469} C_VEL
LIN {X 0,Y 482.152,Z 621.424,A -85,B 0,C 180,E1 21365.431,E2 21365.431} C_VEL
LIN {X 0,Y 481.085,Z 627.928,A -85,B 0,C 180,E1 21365.323,E2 21365.323} C_VEL
LIN {X 0,Y 479.076,Z 661.98,A -85,B 0,C 180,E1 21364.372,E2 21364.372} C_VEL
LIN {X 0,Y 477.368,Z 684.08,A -85,B 0,C 180,E1 21363.524,E2 21363.524} C_VEL
LIN {X 0,Y 475.188,Z 705.766,A -85,B 0,C 180,E1 21362.451,E2 21362.451} C_VEL
LIN {X 0,Y 472.71,Z 725.9,A -85,B 0,C 180,E1 21361.214,E2 21361.214} C_VEL
LIN {X 0,Y 469.934,Z 745.461,A -85,B 0,C 180,E1 21359.759,E2 21359.759} C_VEL
LIN {X 0,Y 467.104,Z 763.42,A -85,B 0,C 180,E1 21358.165,E2 21358.165} C_VEL
LIN {X 0,Y 464.147,Z 780.829,A -85,B 0,C 180,E1 21356.34,E2 21356.34} C_VEL
LIN {X 0,Y 461.249,Z 797.096,A -85,B 0,C 180,E1 21354.323,E2 21354.323} C_VEL
LIN {X 0,Y 458.555,Z 811.859,A -85,B 0,C 180,E1 21352.162,E2 21352.162} C_VEL
LIN {X 0,Y 456.146,Z 825.154,A -85,B 0,C 180,E1 21349.863,E2 21349.863} C_VEL
LIN {X 0,Y 454.078,Z 836.979,A -85,B 0,C 180,E1 21347.426,E2 21347.426} C_VEL
LIN {X 0,Y 452.378,Z 847.3,A -85,B 0,C 180,E1 21344.856,E2 21344.856} C_VEL
LIN {X 0,Y 451.083,Z 856.031,A -85,B 0,C 180,E1 21342.157,E2 21342.157} C_VEL
LIN {X 0,Y 450.214,Z 862.595,A -85,B 0,C 180,E1 21339.566,E2 21339.566} C_VEL
LIN {X 0,Y 449.668,Z 867.666,A -85,B 0,C 180,E1 21336.897,E2 21336.897} C_VEL
LIN {X 0,Y 449.371,Z 871.007,A -85,B 0,C 180,E1 21334.339,E2 21334.339} C_VEL
LIN {X 0,Y 449.224,Z 872.865,A -85,B 0,C 180,E1 21331.658,E2 21331.658} C_VEL
LIN {X 0,Y 449.198,Z 873.077,A -85,B 0,C 180,E1 21329.107,E2 21329.107} C_VEL
LIN {X 0,Y 449.3,Z 871.752,A -85,B 0,C 180,E1 21326.428,E2 21326.428} C_VEL
LIN {X 0,Y 449.556,Z 868.955,A -85,B 0,C 180,E1 21323.832,E2 21323.832} C_VEL
LIN {X 0,Y 450.042,Z 864.162,A -85,B 0,C 180,E1 21321.053,E2 21321.053} C_VEL
LIN {X 0,Y 450.791,Z 858.057,A -85,B 0,C 180,E1 21318.485,E2 21318.485} C_VEL
LIN {X 0,Y 451.971,Z 849.84,A -85,B 0,C 180,E1 21315.785,E2 21315.785} C_VEL
LIN {X 0,Y 453.537,Z 840.114,A -85,B 0,C 180,E1 21313.213,E2 21313.213} C_VEL
LIN {X 0,Y 455.484,Z 828.952,A -85,B 0,C 180,E1 21310.775,E2 21310.775} C_VEL
LIN {X 0,Y 457.768,Z 816.401,A -85,B 0,C 180,E1 21308.472,E2 21308.472} C_VEL
LIN {X 0,Y 460.491,Z 801.535,A -85,B 0,C 180,E1 21306.18,E2 21306.18} C_VEL
LIN {X 0,Y 463.393,Z 785.44,A -85,B 0,C 180,E1 21304.091,E2 21304.091} C_VEL
LIN {X 0,Y 466.333,Z 768.344,A -85,B 0,C 180,E1 21302.216,E2 21302.216} C_VEL
LIN {X 0,Y 469.068,Z 751.399,A -85,B 0,C 180,E1 21300.641,E2 21300.641} C_VEL
LIN {X 0,Y 471.842,Z 732.449,A -85,B 0,C 180,E1 21299.148,E2 21299.148} C_VEL
LIN {X 0,Y 474.38,Z 712.797,A -85,B 0,C 180,E1 21297.858,E2 21297.858} C_VEL
LIN {X 0,Y 476.62,Z 692.451,A -85,B 0,C 180,E1 21296.765,E2 21296.765} C_VEL
LIN {X 0,Y 478.464,Z 671.503,A -85,B 0,C 180,E1 21295.867,E2 21295.867} C_VEL
LIN {X 0,Y 479.862,Z 649.328,A -85,B 0,C 180,E1 21295.144,E2 21295.144} C_VEL
LIN {X 0,Y 482.942,Z 603.252,A -85,B 0,C 180,E1 21293.985,E2 21293.985} C_VEL
LIN {X 0,Y 487.734,Z 535.64,A -85,B 0,C 180,E1 21292.504,E2 21292.504} C_VEL
LIN {X 0,Y 491.458,Z 471.348,A -85,B 0,C 180,E1 21291.284,E2 21291.284} C_VEL
LIN {X 0,Y 494.698,Z 393.121,A -85,B 0,C 180,E1 21290.029,E2 21290.029} C_VEL
LIN {X 0,Y 495.169,Z 382.888,A -85,B 0,C 180,E1 21289.86,E2 21289.86} C_VEL
LIN {X 0,Y 499.455,Z 363.438,A -85,B 0,C 180,E1 21289.108,E2 21289.108} C_VEL
LIN {X 0,Y 499.819,Z 329.349,A -85,B 0,C 180,E1 21286.735,E2 21286.735} C_VEL
LIN {X 0,Y 492.328,Z 309.141,A -85,B 0,C 180,E1 21284.237,E2 21284.237} C_VEL
LIN {X 0,Y 484.713,Z 291.025,A -85,B 0,C 180,E1 21281.782,E2 21281.782} C_VEL
LIN {X 0,Y 477.071,Z 275.122,A -85,B 0,C 180,E1 21279.424,E2 21279.424} C_VEL
LIN {X 0,Y 470.415,Z 262.693,A -85,B 0,C 180,E1 21277.439,E2 21277.439} C_VEL
LIN {X 0,Y 464.9,Z 253.177,A -85,B 0,C 180,E1 21275.804,E2 21275.804} C_VEL
LIN {X 0,Y 462.135,Z 248.659,A -85,B 0,C 180,E1 21274.985,E2 21274.985} C_VEL
LIN {X 0,Y 459.823,Z 244.742,A -85,B 0,C 180,E1 21274.278,E2 21274.278} C_VEL
LIN {X 0,Y 457.513,Z 240.985,A -85,B 0,C 180,E1 21273.568,E2 21273.568} C_VEL
LIN {X 0,Y 456.303,Z 239.305,A -85,B 0,C 180,E1 21273.218,E2 21273.218} C_VEL
LIN {X 0,Y 454.022,Z 235.539,A -85,B 0,C 180,E1 21272.504,E2 21272.504} C_VEL
LIN {X 0,Y 453.254,Z 234.387,A -85,B 0,C 180,E1 21272.267,E2 21272.267} C_VEL
LIN {X 0,Y 451.199,Z 231.945,A -85,B 0,C 180,E1 21271.683,E2 21271.683} C_VEL
LIN {X 0,Y 450.296,Z 229.13,A -85,B 0,C 180,E1 21271.252,E2 21271.252} C_VEL
LIN {X 0,Y 450.293,Z 229.11,A -85,B 0,C 180,E1 21267.508,E2 21267.508} C_VEL
LIN {X 0,Y 450.286,Z 229.098,A -85,B 0,C 180,E1 21263.812,E2 21263.812} C_VEL
LIN {X 0,Y 450.291,Z 229.127,A -85,B 0,C 180,E1 21260.067,E2 21260.067} C_VEL
LIN {X 0,Y 450.291,Z 229.116,A -85,B 0,C 180,E1 21256.38,E2 21256.38} C_VEL
LIN {X 0,Y 450.288,Z 229.092,A -85,B 0,C 180,E1 21252.699,E2 21252.699} C_VEL
LIN {X 0,Y 450.295,Z 229.139,A -85,B 0,C 180,E1 21248.942,E2 21248.942} C_VEL
LIN {X 0,Y 450.283,Z 229.094,A -85,B 0,C 180,E1 21245.224,E2 21245.224} C_VEL
LIN {X 0,Y 450.278,Z 229.126,A -85,B 0,C 180,E1 21241.527,E2 21241.527} C_VEL
LIN {X 0,Y 450.274,Z 229.113,A -85,B 0,C 180,E1 21237.709,E2 21237.709} C_VEL
LIN {X 0,Y 450.283,Z 229.099,A -85,B 0,C 180,E1 21234.009,E2 21234.009} C_VEL
LIN {X 0,Y 450.294,Z 229.133,A -85,B 0,C 180,E1 21230.284,E2 21230.284} C_VEL
LIN {X 0,Y 450.3,Z 229.139,A -85,B 0,C 180,E1 21226.517,E2 21226.517} C_VEL
LIN {X 0,Y 450.292,Z 229.142,A -85,B 0,C 180,E1 21222.823,E2 21222.823} C_VEL
LIN {X 0,Y 450.271,Z 229.136,A -85,B 0,C 180,E1 21219.188,E2 21219.188} C_VEL
LIN {X 0,Y 450.313,Z 229.351,A -85,B 0,C 180,E1 21215.934,E2 21215.934} C_VEL
LIN {X 0,Y 451.415,Z 232.38,A -85,B 0,C 180,E1 21215.391,E2 21215.391} C_VEL
LIN {X 0,Y 452.816,Z 234.512,A -85,B 0,C 180,E1 21214.915,E2 21214.915} C_VEL
LIN {X 0,Y 460.155,Z 248.689,A -85,B 0,C 180,E1 21212.148,E2 21212.148} C_VEL
LIN {X 0,Y 468.901,Z 265.678,A -85,B 0,C 180,E1 21209.075,E2 21209.075} C_VEL
LIN {X 0,Y 478.993,Z 285.851,A -85,B 0,C 180,E1 21205.755,E2 21205.755} C_VEL
LIN {X 0,Y 489.169,Z 306.954,A -85,B 0,C 180,E1 21202.621,E2 21202.621} C_VEL
LIN {X 0,Y 496.135,Z 321.396,A -85,B 0,C 180,E1 21200.667,E2 21200.667} C_VEL
LIN {X 0,Y 504.323,Z 334.524,A -85,B 0,C 180,E1 21199.582,E2 21199.582} C_VEL
LIN {X 0,Y 505.676,Z 351.379,A -85,B 0,C 180,E1 21199.07,E2 21199.07} C_VEL
LIN {X 0,Y 493.439,Z 594.424,A -85,B 0,C 180,E1 21194.823,E2 21194.823} C_VEL
LIN {X 0,Y 489.052,Z 693.147,A -85,B 0,C 180,E1 21193.101,E2 21193.101} C_VEL
LIN {X 0,Y 487.064,Z 717.705,A -85,B 0,C 180,E1 21192.48,E2 21192.48} C_VEL
LIN {X 0,Y 484.689,Z 741.475,A -85,B 0,C 180,E1 21191.687,E2 21191.687} C_VEL
LIN {X 0,Y 482.008,Z 763.641,A -85,B 0,C 180,E1 21190.744,E2 21190.744} C_VEL
LIN {X 0,Y 478.771,Z 787.263,A -85,B 0,C 180,E1 21189.521,E2 21189.521} C_VEL
LIN {X 0,Y 475.64,Z 807.713,A -85,B 0,C 180,E1 21188.25,E2 21188.25} C_VEL
LIN {X 0,Y 471.802,Z 830.773,A -85,B 0,C 180,E1 21186.55,E2 21186.55} C_VEL
LIN {X 0,Y 468.306,Z 850.667,A -85,B 0,C 180,E1 21184.83,E2 21184.83} C_VEL
LIN {X 0,Y 464.826,Z 869.705,A -85,B 0,C 180,E1 21182.904,E2 21182.904} C_VEL
LIN {X 0,Y 461.569,Z 887.432,A -85,B 0,C 180,E1 21180.853,E2 21180.853} C_VEL
LIN {X 0,Y 458.56,Z 903.615,A -85,B 0,C 180,E1 21178.666,E2 21178.666} C_VEL
LIN {X 0,Y 455.749,Z 919.662,A -85,B 0,C 180,E1 21176.191,E2 21176.191} C_VEL
LIN {X 0,Y 453.421,Z 933.611,A -85,B 0,C 180,E1 21173.662,E2 21173.662} C_VEL
LIN {X 0,Y 451.558,Z 946.259,A -85,B 0,C 180,E1 21171.021,E2 21171.021} C_VEL
LIN {X 0,Y 450.159,Z 957.389,A -85,B 0,C 180,E1 21168.251,E2 21168.251} C_VEL
LIN {X 0,Y 449.189,Z 967.193,A -85,B 0,C 180,E1 21165.361,E2 21165.361} C_VEL
LIN {X 0,Y 448.675,Z 974.712,A -85,B 0,C 180,E1 21162.615,E2 21162.615} C_VEL
LIN {X 0,Y 448.445,Z 981.014,A -85,B 0,C 180,E1 21159.756,E2 21159.756} C_VEL
LIN {X 0,Y 448.43,Z 985.494,A -85,B 0,C 180,E1 21156.916,E2 21156.916} C_VEL
LIN {X 0,Y 448.492,Z 988.15,A -85,B 0,C 180,E1 21154.475,E2 21154.475} C_VEL
LIN {X 0,Y 448.566,Z 989.821,A -85,B 0,C 180,E1 21151.66,E2 21151.66} C_VEL
LIN {X 0,Y 448.582,Z 989.831,A -85,B 0,C 180,E1 21148.978,E2 21148.978} C_VEL
LIN {X 0,Y 448.552,Z 988.674,A -85,B 0,C 180,E1 21146.549,E2 21146.549} C_VEL
LIN {X 0,Y 448.472,Z 985.962,A -85,B 0,C 180,E1 21143.728,E2 21143.728} C_VEL
LIN {X 0,Y 448.462,Z 981.519,A -85,B 0,C 180,E1 21140.892,E2 21140.892} C_VEL
LIN {X 0,Y 448.59,Z 976.15,A -85,B 0,C 180,E1 21138.297,E2 21138.297} C_VEL
LIN {X 0,Y 449.049,Z 968.252,A -85,B 0,C 180,E1 21135.295,E2 21135.295} C_VEL
LIN {X 0,Y 449.779,Z 959.77,A -85,B 0,C 180,E1 21132.669,E2 21132.669} C_VEL
LIN {X 0,Y 451.063,Z 948.711,A -85,B 0,C 180,E1 21129.769,E2 21129.769} C_VEL
LIN {X 0,Y 452.845,Z 936.106,A -85,B 0,C 180,E1 21126.994,E2 21126.994} C_VEL
LIN {X 0,Y 455.38,Z 920.711,A -85,B 0,C 180,E1 21124.09,E2 21124.09} C_VEL
LIN {X 0,Y 458.179,Z 905.313,A -85,B 0,C 180,E1 21121.592,E2 21121.592} C_VEL
LIN {X 0,Y 461.612,Z 887.583,A -85,B 0,C 180,E1 21119.112,E2 21119.112} C_VEL
LIN {X 0,Y 465.255,Z 869.575,A -85,B 0,C 180,E1 21116.915,E2 21116.915} C_VEL
LIN {X 0,Y 469.16,Z 850.023,A -85,B 0,C 180,E1 21114.87,E2 21114.87} C_VEL
LIN {X 0,Y 473.357,Z 829.218,A -85,B 0,C 180,E1 21112.984,E2 21112.984} C_VEL
LIN {X 0,Y 477.469,Z 807.865,A -85,B 0,C 180,E1 21111.331,E2 21111.331} C_VEL
LIN {X 0,Y 481.578,Z 785.351,A -85,B 0,C 180,E1 21109.858,E2 21109.858} C_VEL
LIN {X 0,Y 485.477,Z 762.75,A -85,B 0,C 180,E1 21108.613,E2 21108.613} C_VEL
LIN {X 0,Y 489.041,Z 739.355,A -85,B 0,C 180,E1 21107.568,E2 21107.568} C_VEL
LIN {X 0,Y 492.468,Z 713.955,A -85,B 0,C 180,E1 21106.67,E2 21106.67} C_VEL
LIN {X 0,Y 495.235,Z 689.22,A -85,B 0,C 180,E1 21106.009,E2 21106.009} C_VEL
LIN {X 0,Y 502.415,Z 606.101,A -85,B 0,C 180,E1 21104.283,E2 21104.283} C_VEL
LIN {X 0,Y 509.652,Z 543.883,A -85,B 0,C 180,E1 21102.893,E2 21102.893} C_VEL
LIN {X 0,Y 518.608,Z 484.008,A -85,B 0,C 180,E1 21101.477,E2 21101.477} C_VEL
LIN {X 0,Y 529.824,Z 424.254,A -85,B 0,C 180,E1 21100.048,E2 21100.048} C_VEL
LIN {X 0,Y 530.345,Z 421.728,A -85,B 0,C 180,E1 21099.978,E2 21099.978} C_VEL
LIN {X 0,Y 525.481,Z 439.424,A -85,B 0,C 180,E1 21098.653,E2 21098.653} C_VEL
LIN {X 0,Y 521.194,Z 459.651,A -85,B 0,C 180,E1 21097.309,E2 21097.309} C_VEL
LIN {X 0,Y 517.046,Z 484.385,A -85,B 0,C 180,E1 21095.862,E2 21095.862} C_VEL
LIN {X 0,Y 512.915,Z 514.472,A -85,B 0,C 180,E1 21094.316,E2 21094.316} C_VEL
LIN {X 0,Y 511.601,Z 522.309,A -85,B 0,C 180,E1 21094.061,E2 21094.061} C_VEL
LIN {X 0,Y 494.044,Z 627.424,A -85,B 0,C 180,E1 21091.033,E2 21091.033} C_VEL
LIN {X 0,Y 484.529,Z 693.436,A -85,B 0,C 180,E1 21089.026,E2 21089.026} C_VEL
LIN {X 0,Y 480.673,Z 717.867,A -85,B 0,C 180,E1 21088.042,E2 21088.042} C_VEL
LIN {X 0,Y 476.883,Z 740.991,A -85,B 0,C 180,E1 21086.862,E2 21086.862} C_VEL
LIN {X 0,Y 473.152,Z 763.244,A -85,B 0,C 180,E1 21085.471,E2 21085.471} C_VEL
LIN {X 0,Y 469.661,Z 783.67,A -85,B 0,C 180,E1 21083.927,E2 21083.927} C_VEL
LIN {X 0,Y 466.419,Z 802.263,A -85,B 0,C 180,E1 21082.233,E2 21082.233} C_VEL
LIN {X 0,Y 463.679,Z 817.604,A -85,B 0,C 180,E1 21080.579,E2 21080.579} C_VEL
LIN {X 0,Y 461.038,Z 832.136,A -85,B 0,C 180,E1 21078.722,E2 21078.722} C_VEL
LIN {X 0,Y 458.61,Z 845.081,A -85,B 0,C 180,E1 21076.726,E2 21076.726} C_VEL
LIN {X 0,Y 456.552,Z 855.769,A -85,B 0,C 180,E1 21074.717,E2 21074.717} C_VEL
LIN {X 0,Y 454.829,Z 864.486,A -85,B 0,C 180,E1 21072.7,E2 21072.7} C_VEL
LIN {X 0,Y 453.255,Z 872.152,A -85,B 0,C 180,E1 21070.422,E2 21070.422} C_VEL
LIN {X 0,Y 452.041,Z 877.742,A -85,B 0,C 180,E1 21068.138,E2 21068.138} C_VEL
LIN {X 0,Y 451.139,Z 881.424,A -85,B 0,C 180,E1 21065.852,E2 21065.852} C_VEL
LIN {X 0,Y 450.515,Z 883.217,A -85,B 0,C 180,E1 21063.69,E2 21063.69} C_VEL
LIN {X 0,Y 450.074,Z 883.39,A -85,B 0,C 180,E1 21061.4,E2 21061.4} C_VEL
LIN {X 0,Y 449.815,Z 881.823,A -85,B 0,C 180,E1 21059.108,E2 21059.108} C_VEL
LIN {X 0,Y 449.716,Z 878.498,A -85,B 0,C 180,E1 21056.814,E2 21056.814} C_VEL
LIN {X 0,Y 449.795,Z 873.387,A -85,B 0,C 180,E1 21054.515,E2 21054.515} C_VEL
LIN {X 0,Y 450.067,Z 866.52,A -85,B 0,C 180,E1 21052.247,E2 21052.247} C_VEL
LIN {X 0,Y 450.558,Z 857.917,A -85,B 0,C 180,E1 21050.032,E2 21050.032} C_VEL
LIN {X 0,Y 451.318,Z 847.405,A -85,B 0,C 180,E1 21047.85,E2 21047.85} C_VEL
LIN {X 0,Y 452.311,Z 835.396,A -85,B 0,C 180,E1 21045.796,E2 21045.796} C_VEL
LIN {X 0,Y 453.613,Z 820.956,A -85,B 0,C 180,E1 21043.743,E2 21043.743} C_VEL
LIN {X 0,Y 455.089,Z 805.309,A -85,B 0,C 180,E1 21041.887,E2 21041.887} C_VEL
LIN {X 0,Y 456.753,Z 787.953,A -85,B 0,C 180,E1 21040.165,E2 21040.165} C_VEL
LIN {X 0,Y 458.462,Z 769.351,A -85,B 0,C 180,E1 21038.635,E2 21038.635} C_VEL
LIN {X 0,Y 460.196,Z 749.84,A -85,B 0,C 180,E1 21037.315,E2 21037.315} C_VEL
LIN {X 0,Y 461.88,Z 729.249,A -85,B 0,C 180,E1 21036.188,E2 21036.188} C_VEL
LIN {X 0,Y 463.467,Z 707.122,A -85,B 0,C 180,E1 21035.24,E2 21035.24} C_VEL
LIN {X 0,Y 464.819,Z 685.119,A -85,B 0,C 180,E1 21034.548,E2 21034.548} C_VEL
LIN {X 0,Y 473.257,Z 502.719,A -85,B 0,C 180,E1 21030.692,E2 21030.692} C_VEL
LIN {X 0,Y 468.265,Z 442.042,A -85,B 0,C 180,E1 21028.85,E2 21028.85} C_VEL
LIN {X 0,Y 473.624,Z 389.762,A -85,B 0,C 180,E1 21024.787,E2 21024.787} C_VEL
LIN {X 0,Y 479.379,Z 338.841,A -85,B 0,C 180,E1 21020.802,E2 21020.802} C_VEL
LIN {X 0,Y 482.929,Z 309.227,A -85,B 0,C 180,E1 21018.468,E2 21018.468} C_VEL
LIN {X 0,Y 480.743,Z 303.161,A -85,B 0,C 180,E1 21017.713,E2 21017.713} C_VEL
LIN {X 0,Y 482.802,Z 303.744,A -85,B 0,C 180,E1 21017.373,E2 21017.373} C_VEL
LIN {X 0,Y 490.134,Z 303.685,A -85,B 0,C 180,E1 21016.366,E2 21016.366} C_VEL
LIN {X 0,Y 497.91,Z 324.114,A -85,B 0,C 180,E1 21013.785,E2 21013.785} C_VEL
LIN {X 0,Y 499.866,Z 330.008,A -85,B 0,C 180,E1 21013.104,E2 21013.104} C_VEL
LIN {X 0,Y 499.283,Z 364.047,A -85,B 0,C 180,E1 21010.758,E2 21010.758} C_VEL
LIN {X 0,Y 494.952,Z 384.388,A -85,B 0,C 180,E1 21010.005,E2 21010.005} C_VEL
LIN {X 0,Y 491.542,Z 468.475,A -85,B 0,C 180,E1 21008.669,E2 21008.669} C_VEL
LIN {X 0,Y 487.771,Z 534.231,A -85,B 0,C 180,E1 21007.426,E2 21007.426} C_VEL
LIN {X 0,Y 482.681,Z 606.165,A -85,B 0,C 180,E1 21005.85,E2 21005.85} C_VEL
LIN {X 0,Y 481.085,Z 627.928,A -85,B 0,C 180,E1 21005.323,E2 21005.323} C_VEL
LIN {X 0,Y 479.763,Z 635.517,A -85,B 0,C 180,E1 21005.2,E2 21005.2} C_VEL
LIN {X 0,Y 473.715,Z 654.685,A -85,B 0,C 180,E1 21005.098,E2 21005.098} C_VEL
LIN {X 0,Y 472.525,Z 662.213,A -85,B 0,C 180,E1 21004.928,E2 21004.928} C_VEL
LIN {X 0,Y 470.817,Z 683.781,A -85,B 0,C 180,E1 21004.102,E2 21004.102} C_VEL
LIN {X 0,Y 468.734,Z 704.222,A -85,B 0,C 180,E1 21003.099,E2 21003.099} C_VEL
LIN {X 0,Y 466.184,Z 724.726,A -85,B 0,C 180,E1 21001.858,E2 21001.858} C_VEL
LIN {X 0,Y 463.318,Z 744.487,A -85,B 0,C 180,E1 21000.401,E2 21000.401} C_VEL
LIN {X 0,Y 460.204,Z 763.725,A -85,B 0,C 180,E1 20998.697,E2 20998.697} C_VEL
LIN {X 0,Y 457.019,Z 781.761,A -85,B 0,C 180,E1 20996.789,E2 20996.789} C_VEL
LIN {X 0,Y 453.984,Z 798.079,A -85,B 0,C 180,E1 20994.738,E2 20994.738} C_VEL
LIN {X 0,Y 451.166,Z 812.861,A -85,B 0,C 180,E1 20992.545,E2 20992.545} C_VEL
LIN {X 0,Y 448.637,Z 826.157,A -85,B 0,C 180,E1 20990.21,E2 20990.21} C_VEL
LIN {X 0,Y 446.458,Z 837.988,A -85,B 0,C 180,E1 20987.733,E2 20987.733} C_VEL
LIN {X 0,Y 444.658,Z 848.297,A -85,B 0,C 180,E1 20985.12,E2 20985.12} C_VEL
LIN {X 0,Y 443.284,Z 857.031,A -85,B 0,C 180,E1 20982.374,E2 20982.374} C_VEL
LIN {X 0,Y 442.358,Z 863.547,A -85,B 0,C 180,E1 20979.76,E2 20979.76} C_VEL
LIN {X 0,Y 441.767,Z 868.671,A -85,B 0,C 180,E1 20977.021,E2 20977.021} C_VEL
LIN {X 0,Y 441.434,Z 872.12,A -85,B 0,C 180,E1 20974.287,E2 20974.287} C_VEL
LIN {X 0,Y 441.285,Z 873.933,A -85,B 0,C 180,E1 20971.558,E2 20971.558} C_VEL
LIN {X 0,Y 441.265,Z 874.056,A -85,B 0,C 180,E1 20968.961,E2 20968.961} C_VEL
LIN {X 0,Y 441.381,Z 872.641,A -85,B 0,C 180,E1 20966.233,E2 20966.233} C_VEL
LIN {X 0,Y 441.658,Z 869.817,A -85,B 0,C 180,E1 20963.631,E2 20963.631} C_VEL
LIN {X 0,Y 442.172,Z 865.168,A -85,B 0,C 180,E1 20960.892,E2 20960.892} C_VEL
LIN {X 0,Y 442.974,Z 859.061,A -85,B 0,C 180,E1 20958.279,E2 20958.279} C_VEL
LIN {X 0,Y 444.159,Z 851.277,A -85,B 0,C 180,E1 20955.663,E2 20955.663} C_VEL
LIN {X 0,Y 445.794,Z 841.651,A -85,B 0,C 180,E1 20953.047,E2 20953.047} C_VEL
LIN {X 0,Y 447.823,Z 830.601,A -85,B 0,C 180,E1 20950.568,E2 20950.568} C_VEL
LIN {X 0,Y 450.273,Z 817.754,A -85,B 0,C 180,E1 20948.16,E2 20948.16} C_VEL
LIN {X 0,Y 453.021,Z 803.399,A -85,B 0,C 180,E1 20945.9,E2 20945.9} C_VEL
LIN {X 0,Y 456.029,Z 787.439,A -85,B 0,C 180,E1 20943.781,E2 20943.781} C_VEL
LIN {X 0,Y 459.015,Z 770.826,A -85,B 0,C 180,E1 20941.913,E2 20941.913} C_VEL
LIN {X 0,Y 461.904,Z 753.768,A -85,B 0,C 180,E1 20940.283,E2 20940.283} C_VEL
LIN {X 0,Y 464.9,Z 734.209,A -85,B 0,C 180,E1 20938.707,E2 20938.707} C_VEL
LIN {X 0,Y 467.548,Z 714.477,A -85,B 0,C 180,E1 20937.39,E2 20937.39} C_VEL
LIN {X 0,Y 469.84,Z 694.497,A -85,B 0,C 180,E1 20936.296,E2 20936.296} C_VEL
LIN {X 0,Y 471.765,Z 673.569,A -85,B 0,C 180,E1 20935.379,E2 20935.379} C_VEL
LIN {X 0,Y 473.232,Z 651.389,A -85,B 0,C 180,E1 20934.638,E2 20934.638} C_VEL
LIN {X 0,Y 476.293,Z 606.899,A -85,B 0,C 180,E1 20933.49,E2 20933.49} C_VEL
LIN {X 0,Y 481.206,Z 540.255,A -85,B 0,C 180,E1 20932.002,E2 20932.002} C_VEL
LIN {X 0,Y 485.108,Z 475.854,A -85,B 0,C 180,E1 20930.756,E2 20930.756} C_VEL
LIN {X 0,Y 488.427,Z 399.113,A -85,B 0,C 180,E1 20929.509,E2 20929.509} C_VEL
LIN {X 0,Y 489.027,Z 385.666,A -85,B 0,C 180,E1 20929.289,E2 20929.289} C_VEL
LIN {X 0,Y 493.565,Z 365.343,A -85,B 0,C 180,E1 20928.513,E2 20928.513} C_VEL
LIN {X 0,Y 493.921,Z 333.3,A -85,B 0,C 180,E1 20926.279,E2 20926.279} C_VEL
LIN {X 0,Y 486.305,Z 312.723,A -85,B 0,C 180,E1 20923.698,E2 20923.698} C_VEL
LIN {X 0,Y 478.6,Z 294.408,A -85,B 0,C 180,E1 20921.155,E2 20921.155} C_VEL
LIN {X 0,Y 470.59,Z 277.843,A -85,B 0,C 180,E1 20918.659,E2 20918.659} C_VEL
LIN {X 0,Y 463.675,Z 264.985,A -85,B 0,C 180,E1 20916.526,E2 20916.526} C_VEL
LIN {X 0,Y 457.471,Z 254.543,A -85,B 0,C 180,E1 20914.631,E2 20914.631} C_VEL
LIN {X 0,Y 455.192,Z 250.74,A -85,B 0,C 180,E1 20913.914,E2 20913.914} C_VEL
LIN {X 0,Y 452.103,Z 245.816,A -85,B 0,C 180,E1 20912.961,E2 20912.961} C_VEL
LIN {X 0,Y 449.837,Z 242.202,A -85,B 0,C 180,E1 20912.24,E2 20912.24} C_VEL
LIN {X 0,Y 448.675,Z 240.567,A -85,B 0,C 180,E1 20911.882,E2 20911.882} C_VEL
LIN {X 0,Y 446.433,Z 237.103,A -85,B 0,C 180,E1 20911.157,E2 20911.157} C_VEL
LIN {X 0,Y 445.754,Z 235.733,A -85,B 0,C 180,E1 20910.909,E2 20910.909} C_VEL
LIN {X 0,Y 443.354,Z 233.096,A -85,B 0,C 180,E1 20910.194,E2 20910.194} C_VEL
LIN {X 0,Y 442.354,Z 230.106,A -85,B 0,C 180,E1 20909.711,E2 20909.711} C_VEL
LIN {X 0,Y 442.354,Z 230.128,A -85,B 0,C 180,E1 20905.865,E2 20905.865} C_VEL
LIN {X 0,Y 442.354,Z 230.101,A -85,B 0,C 180,E1 20902.038,E2 20902.038} C_VEL
LIN {X 0,Y 442.351,Z 230.08,A -85,B 0,C 180,E1 20898.311,E2 20898.311} C_VEL
LIN {X 0,Y 442.353,Z 230.117,A -85,B 0,C 180,E1 20894.531,E2 20894.531} C_VEL
LIN {X 0,Y 442.351,Z 230.097,A -85,B 0,C 180,E1 20890.682,E2 20890.682} C_VEL
LIN {X 0,Y 442.357,Z 230.083,A -85,B 0,C 180,E1 20886.881,E2 20886.881} C_VEL
LIN {X 0,Y 442.349,Z 230.128,A -85,B 0,C 180,E1 20883.11,E2 20883.11} C_VEL
LIN {X 0,Y 442.337,Z 230.076,A -85,B 0,C 180,E1 20879.352,E2 20879.352} C_VEL
LIN {X 0,Y 442.336,Z 230.128,A -85,B 0,C 180,E1 20875.592,E2 20875.592} C_VEL
LIN {X 0,Y 442.334,Z 230.084,A -85,B 0,C 180,E1 20871.813,E2 20871.813} C_VEL
LIN {X 0,Y 442.352,Z 230.13,A -85,B 0,C 180,E1 20868.13,E2 20868.13} C_VEL
LIN {X 0,Y 442.361,Z 230.116,A -85,B 0,C 180,E1 20864.346,E2 20864.346} C_VEL
LIN {X 0,Y 442.36,Z 230.122,A -85,B 0,C 180,E1 20860.593,E2 20860.593} C_VEL
LIN {X 0,Y 442.336,Z 230.175,A -85,B 0,C 180,E1 20857.19,E2 20857.19} C_VEL
LIN {X 0,Y 443.713,Z 233.671,A -85,B 0,C 180,E1 20856.514,E2 20856.514} C_VEL
LIN {X 0,Y 444.82,Z 235.229,A -85,B 0,C 180,E1 20856.133,E2 20856.133} C_VEL
LIN {X 0,Y 446.588,Z 238.926,A -85,B 0,C 180,E1 20855.389,E2 20855.389} C_VEL
LIN {X 0,Y 452.364,Z 249.899,A -85,B 0,C 180,E1 20853.197,E2 20853.197} C_VEL
LIN {X 0,Y 459.607,Z 263.997,A -85,B 0,C 180,E1 20850.549,E2 20850.549} C_VEL
LIN {X 0,Y 469.317,Z 283.159,A -85,B 0,C 180,E1 20847.238,E2 20847.238} C_VEL
LIN {X 0,Y 479.486,Z 304.083,A -85,B 0,C 180,E1 20843.98,E2 20843.98} C_VEL
LIN {X 0,Y 488.185,Z 322.254,A -85,B 0,C 180,E1 20841.434,E2 20841.434} C_VEL
LIN {X 0,Y 498.33,Z 338.535,A -85,B 0,C 180,E1 20840.053,E2 20840.053} C_VEL
LIN {X 0,Y 499.433,Z 352.494,A -85,B 0,C 180,E1 20839.632,E2 20839.632} C_VEL
LIN {X 0,Y 486.734,Z 594.185,A -85,B 0,C 180,E1 20835.337,E2 20835.337} C_VEL
LIN {X 0,Y 482.147,Z 693.173,A -85,B 0,C 180,E1 20833.579,E2 20833.579} C_VEL
LIN {X 0,Y 480.107,Z 717.55,A -85,B 0,C 180,E1 20832.951,E2 20832.951} C_VEL
LIN {X 0,Y 477.638,Z 741.517,A -85,B 0,C 180,E1 20832.139,E2 20832.139} C_VEL
LIN {X 0,Y 474.804,Z 764.239,A -85,B 0,C 180,E1 20831.155,E2 20831.155} C_VEL
LIN {X 0,Y 471.297,Z 788.852,A -85,B 0,C 180,E1 20829.845,E2 20829.845} C_VEL
LIN {X 0,Y 468.02,Z 809.633,A -85,B 0,C 180,E1 20828.519,E2 20828.519} C_VEL
LIN {X 0,Y 464.382,Z 830.763,A -85,B 0,C 180,E1 20826.922,E2 20826.922} C_VEL
LIN {X 0,Y 460.669,Z 851.372,A -85,B 0,C 180,E1 20825.113,E2 20825.113} C_VEL
LIN {X 0,Y 457.099,Z 870.27,A -85,B 0,C 180,E1 20823.152,E2 20823.152} C_VEL
LIN {X 0,Y 453.612,Z 888.611,A -85,B 0,C 180,E1 20820.966,E2 20820.966} C_VEL
LIN {X 0,Y 450.609,Z 904.415,A -85,B 0,C 180,E1 20818.777,E2 20818.777} C_VEL
LIN {X 0,Y 447.737,Z 920.352,A -85,B 0,C 180,E1 20816.243,E2 20816.243} C_VEL
LIN {X 0,Y 445.513,Z 933.366,A -85,B 0,C 180,E1 20813.827,E2 20813.827} C_VEL
LIN {X 0,Y 443.525,Z 946.498,A -85,B 0,C 180,E1 20811.005,E2 20811.005} C_VEL
LIN {X 0,Y 442.234,Z 956.556,A -85,B 0,C 180,E1 20808.454,E2 20808.454} C_VEL
LIN {X 0,Y 441.234,Z 966.379,A -85,B 0,C 180,E1 20805.51,E2 20805.51} C_VEL
LIN {X 0,Y 440.71,Z 973.894,A -85,B 0,C 180,E1 20802.713,E2 20802.713} C_VEL
LIN {X 0,Y 440.479,Z 980.191,A -85,B 0,C 180,E1 20799.802,E2 20799.802} C_VEL
LIN {X 0,Y 440.472,Z 984.655,A -85,B 0,C 180,E1 20796.91,E2 20796.91} C_VEL
LIN {X 0,Y 440.544,Z 987.29,A -85,B 0,C 180,E1 20794.426,E2 20794.426} C_VEL
LIN {X 0,Y 440.622,Z 988.907,A -85,B 0,C 180,E1 20791.56,E2 20791.56} C_VEL
LIN {X 0,Y 440.64,Z 988.873,A -85,B 0,C 180,E1 20788.83,E2 20788.83} C_VEL
LIN {X 0,Y 440.591,Z 987.574,A -85,B 0,C 180,E1 20786.226,E2 20786.226} C_VEL
LIN {X 0,Y 440.504,Z 984.504,A -85,B 0,C 180,E1 20783.221,E2 20783.221} C_VEL
LIN {X 0,Y 440.507,Z 980.114,A -85,B 0,C 180,E1 20780.462,E2 20780.462} C_VEL
LIN {X 0,Y 440.672,Z 974.32,A -85,B 0,C 180,E1 20777.685,E2 20777.685} C_VEL
LIN {X 0,Y 441.199,Z 966.109,A -85,B 0,C 180,E1 20774.624,E2 20774.624} C_VEL
LIN {X 0,Y 442.052,Z 957.443,A -85,B 0,C 180,E1 20771.948,E2 20771.948} C_VEL
LIN {X 0,Y 443.569,Z 945.475,A -85,B 0,C 180,E1 20768.858,E2 20768.858} C_VEL
LIN {X 0,Y 445.464,Z 933.249,A -85,B 0,C 180,E1 20766.17,E2 20766.17} C_VEL
LIN {X 0,Y 448.123,Z 918.275,A -85,B 0,C 180,E1 20763.353,E2 20763.353} C_VEL
LIN {X 0,Y 451.347,Z 901.888,A -85,B 0,C 180,E1 20760.686,E2 20760.686} C_VEL
LIN {X 0,Y 454.861,Z 884.689,A -85,B 0,C 180,E1 20758.29,E2 20758.29} C_VEL
LIN {X 0,Y 458.989,Z 865.406,A -85,B 0,C 180,E1 20755.953,E2 20755.953} C_VEL
LIN {X 0,Y 463.108,Z 846.356,A -85,B 0,C 180,E1 20753.965,E2 20753.965} C_VEL
LIN {X 0,Y 467.571,Z 825.15,A -85,B 0,C 180,E1 20752.062,E2 20752.062} C_VEL
LIN {X 0,Y 472.033,Z 803.403,A -85,B 0,C 180,E1 20750.387,E2 20750.387} C_VEL
LIN {X 0,Y 476.407,Z 780.8,A -85,B 0,C 180,E1 20748.934,E2 20748.934} C_VEL
LIN {X 0,Y 480.762,Z 756.468,A -85,B 0,C 180,E1 20747.634,E2 20747.634} C_VEL
LIN {X 0,Y 484.653,Z 732.586,A -85,B 0,C 180,E1 20746.6,E2 20746.6} C_VEL
LIN {X 0,Y 487.681,Z 710.897,A -85,B 0,C 180,E1 20745.858,E2 20745.858} C_VEL
LIN {X 0,Y 490.649,Z 685.393,A -85,B 0,C 180,E1 20745.187,E2 20745.187} C_VEL
LIN {X 0,Y 498.083,Z 609.195,A -85,B 0,C 180,E1 20743.551,E2 20743.551} C_VEL
LIN {X 0,Y 505.934,Z 548.706,A -85,B 0,C 180,E1 20742.162,E2 20742.162} C_VEL
LIN {X 0,Y 515.553,Z 490.353,A -85,B 0,C 180,E1 20740.758,E2 20740.758} C_VEL
LIN {X 0,Y 525.388,Z 441.268,A -85,B 0,C 180,E1 20739.557,E2 20739.557} C_VEL
LIN {X 0,Y 520.306,Z 461.147,A -85,B 0,C 180,E1 20738.218,E2 20738.218} C_VEL
LIN {X 0,Y 515.375,Z 485.401,A -85,B 0,C 180,E1 20736.765,E2 20736.765} C_VEL
LIN {X 0,Y 510.589,Z 514.281,A -85,B 0,C 180,E1 20735.243,E2 20735.243} C_VEL
LIN {X 0,Y 509.603,Z 520.313,A -85,B 0,C 180,E1 20734.989,E2 20734.989} C_VEL
LIN {X 0,Y 490.6,Z 625.827,A -85,B 0,C 180,E1 20731.918,E2 20731.918} C_VEL
LIN {X 0,Y 479.982,Z 693.641,A -85,B 0,C 180,E1 20729.817,E2 20729.817} C_VEL
LIN {X 0,Y 475.83,Z 717.695,A -85,B 0,C 180,E1 20728.833,E2 20728.833} C_VEL
LIN {X 0,Y 471.557,Z 741.406,A -85,B 0,C 180,E1 20727.601,E2 20727.601} C_VEL
LIN {X 0,Y 467.523,Z 763.24,A -85,B 0,C 180,E1 20726.209,E2 20726.209} C_VEL
LIN {X 0,Y 463.727,Z 783.446,A -85,B 0,C 180,E1 20724.66,E2 20724.66} C_VEL
LIN {X 0,Y 460.107,Z 802.686,A -85,B 0,C 180,E1 20722.892,E2 20722.892} C_VEL
LIN {X 0,Y 456.73,Z 820.031,A -85,B 0,C 180,E1 20720.974,E2 20720.974} C_VEL
LIN {X 0,Y 453.819,Z 834.644,A -85,B 0,C 180,E1 20719.031,E2 20719.031} C_VEL
LIN {X 0,Y 451.393,Z 846.564,A -85,B 0,C 180,E1 20717.134,E2 20717.134} C_VEL
LIN {X 0,Y 449.196,Z 857.195,A -85,B 0,C 180,E1 20715.096,E2 20715.096} C_VEL
LIN {X 0,Y 447.195,Z 866.471,A -85,B 0,C 180,E1 20712.874,E2 20712.874} C_VEL
LIN {X 0,Y 445.638,Z 873.434,A -85,B 0,C 180,E1 20710.733,E2 20710.733} C_VEL
LIN {X 0,Y 444.323,Z 878.997,A -85,B 0,C 180,E1 20708.411,E2 20708.411} C_VEL
LIN {X 0,Y 443.386,Z 882.462,A -85,B 0,C 180,E1 20706.214,E2 20706.214} C_VEL
LIN {X 0,Y 442.657,Z 884.395,A -85,B 0,C 180,E1 20703.886,E2 20703.886} C_VEL
LIN {X 0,Y 442.173,Z 884.551,A -85,B 0,C 180,E1 20701.555,E2 20701.555} C_VEL
LIN {X 0,Y 441.888,Z 882.931,A -85,B 0,C 180,E1 20699.222,E2 20699.222} C_VEL
LIN {X 0,Y 441.77,Z 879.587,A -85,B 0,C 180,E1 20696.886,E2 20696.886} C_VEL
LIN {X 0,Y 441.842,Z 874.438,A -85,B 0,C 180,E1 20694.546,E2 20694.546} C_VEL
LIN {X 0,Y 442.121,Z 867.4,A -85,B 0,C 180,E1 20692.201,E2 20692.201} C_VEL
LIN {X 0,Y 442.654,Z 858.321,A -85,B 0,C 180,E1 20689.852,E2 20689.852} C_VEL
LIN {X 0,Y 443.451,Z 847.643,A -85,B 0,C 180,E1 20687.631,E2 20687.631} C_VEL
LIN {X 0,Y 444.491,Z 835.454,A -85,B 0,C 180,E1 20685.54,E2 20685.54} C_VEL
LIN {X 0,Y 445.803,Z 821.309,A -85,B 0,C 180,E1 20683.517,E2 20683.517} C_VEL
LIN {X 0,Y 447.334,Z 805.541,A -85,B 0,C 180,E1 20681.629,E2 20681.629} C_VEL
LIN {X 0,Y 449.056,Z 788.052,A -85,B 0,C 180,E1 20679.878,E2 20679.878} C_VEL
LIN {X 0,Y 450.81,Z 769.422,A -85,B 0,C 180,E1 20678.332,E2 20678.332} C_VEL
LIN {X 0,Y 452.615,Z 749.647,A -85,B 0,C 180,E1 20676.982,E2 20676.982} C_VEL
LIN {X 0,Y 454.354,Z 728.912,A -85,B 0,C 180,E1 20675.837,E2 20675.837} C_VEL
LIN {X 0,Y 455.969,Z 706.942,A -85,B 0,C 180,E1 20674.888,E2 20674.888} C_VEL
LIN {X 0,Y 457.382,Z 684.74,A -85,B 0,C 180,E1 20674.177,E2 20674.177} C_VEL
LIN {X 0,Y 466.116,Z 503.547,A -85,B 0,C 180,E1 20670.256,E2 20670.256} C_VEL
LIN {X 0,Y 461.086,Z 441.386,A -85,B 0,C 180,E1 20668.346,E2 20668.346} C_VEL
LIN {X 0,Y 466.557,Z 390.221,A -85,B 0,C 180,E1 20664.316,E2 20664.316} C_VEL
LIN {X 0,Y 472.538,Z 339.274,A -85,B 0,C 180,E1 20660.28,E2 20660.28} C_VEL
LIN {X 0,Y 475.943,Z 312.332,A -85,B 0,C 180,E1 20658.138,E2 20658.138} C_VEL
LIN {X 0,Y 475.392,Z 310.639,A -85,B 0,C 180,E1 20657.9,E2 20657.9} C_VEL
LIN {X 0,Y 477.295,Z 311.19,A -85,B 0,C 180,E1 20657.58,E2 20657.58} C_VEL
LIN {X 0,Y 485.567,Z 311.009,A -85,B 0,C 180,E1 20656.423,E2 20656.423} C_VEL
LIN {X 0,Y 492.952,Z 330.765,A -85,B 0,C 180,E1 20653.924,E2 20653.924} C_VEL
LIN {X 0,Y 493.948,Z 333.956,A -85,B 0,C 180,E1 20653.556,E2 20653.556} C_VEL
LIN {X 0,Y 493.329,Z 366.026,A -85,B 0,C 180,E1 20651.357,E2 20651.357} C_VEL
LIN {X 0,Y 488.809,Z 387.194,A -85,B 0,C 180,E1 20650.576,E2 20650.576} C_VEL
LIN {X 0,Y 485.308,Z 470.715,A -85,B 0,C 180,E1 20649.236,E2 20649.236} C_VEL
LIN {X 0,Y 481.459,Z 535.724,A -85,B 0,C 180,E1 20647.994,E2 20647.994} C_VEL
LIN {X 0,Y 476.291,Z 606.322,A -85,B 0,C 180,E1 20646.426,E2 20646.426} C_VEL
LIN {X 0,Y 473.186,Z 651.162,A -85,B 0,C 180,E1 20645.268,E2 20645.268} C_VEL
LIN {X 0,Y 472.525,Z 662.213,A -85,B 0,C 180,E1 20644.928,E2 20644.928} C_VEL
LIN {X 0,Y 471.236,Z 669.722,A -85,B 0,C 180,E1 20644.745,E2 20644.745} C_VEL
LIN {X 0,Y 464.678,Z 688.61,A -85,B 0,C 180,E1 20644.398,E2 20644.398} C_VEL
LIN {X 0,Y 463.124,Z 695.785,A -85,B 0,C 180,E1 20644.124,E2 20644.124} C_VEL
LIN {X 0,Y 460.73,Z 715.936,A -85,B 0,C 180,E1 20643.006,E2 20643.006} C_VEL
LIN {X 0,Y 457.992,Z 735.607,A -85,B 0,C 180,E1 20641.672,E2 20641.672} C_VEL
LIN {X 0,Y 454.888,Z 755.12,A -85,B 0,C 180,E1 20640.077,E2 20640.077} C_VEL
LIN {X 0,Y 451.639,Z 773.492,A -85,B 0,C 180,E1 20638.28,E2 20638.28} C_VEL
LIN {X 0,Y 448.465,Z 790.333,A -85,B 0,C 180,E1 20636.324,E2 20636.324} C_VEL
LIN {X 0,Y 445.483,Z 805.483,A -85,B 0,C 180,E1 20634.252,E2 20634.252} C_VEL
LIN {X 0,Y 442.719,Z 819.344,A -85,B 0,C 180,E1 20632.019,E2 20632.019} C_VEL
LIN {X 0,Y 440.066,Z 832.716,A -85,B 0,C 180,E1 20629.448,E2 20629.448} C_VEL
LIN {X 0,Y 437.836,Z 844.411,A -85,B 0,C 180,E1 20626.723,E2 20626.723} C_VEL
LIN {X 0,Y 436.113,Z 854.137,A -85,B 0,C 180,E1 20623.93,E2 20623.93} C_VEL
LIN {X 0,Y 434.937,Z 861.5,A -85,B 0,C 180,E1 20621.269,E2 20621.269} C_VEL
LIN {X 0,Y 434.124,Z 867.452,A -85,B 0,C 180,E1 20618.477,E2 20618.477} C_VEL
LIN {X 0,Y 433.632,Z 871.835,A -85,B 0,C 180,E1 20615.558,E2 20615.558} C_VEL
LIN {X 0,Y 433.405,Z 874.272,A -85,B 0,C 180,E1 20612.909,E2 20612.909} C_VEL
LIN {X 0,Y 433.334,Z 875.196,A -85,B 0,C 180,E1 20610.132,E2 20610.132} C_VEL
LIN {X 0,Y 433.377,Z 874.509,A -85,B 0,C 180,E1 20607.471,E2 20607.471} C_VEL
LIN {X 0,Y 433.61,Z 872.101,A -85,B 0,C 180,E1 20604.575,E2 20604.575} C_VEL
LIN {X 0,Y 434.02,Z 868.367,A -85,B 0,C 180,E1 20601.922,E2 20601.922} C_VEL
LIN {X 0,Y 434.792,Z 862.689,A -85,B 0,C 180,E1 20599.106,E2 20599.106} C_VEL
LIN {X 0,Y 435.932,Z 855.237,A -85,B 0,C 180,E1 20596.335,E2 20596.335} C_VEL
LIN {X 0,Y 437.492,Z 846.246,A -85,B 0,C 180,E1 20593.673,E2 20593.673} C_VEL
LIN {X 0,Y 439.441,Z 835.877,A -85,B 0,C 180,E1 20591.149,E2 20591.149} C_VEL
LIN {X 0,Y 441.886,Z 823.475,A -85,B 0,C 180,E1 20588.635,E2 20588.635} C_VEL
LIN {X 0,Y 444.532,Z 810.383,A -85,B 0,C 180,E1 20586.398,E2 20586.398} C_VEL
LIN {X 0,Y 447.552,Z 795.239,A -85,B 0,C 180,E1 20584.205,E2 20584.205} C_VEL
LIN {X 0,Y 450.668,Z 779.131,A -85,B 0,C 180,E1 20582.23,E2 20582.23} C_VEL
LIN {X 0,Y 453.876,Z 761.355,A -85,B 0,C 180,E1 20580.39,E2 20580.39} C_VEL
LIN {X 0,Y 456.985,Z 742.634,A -85,B 0,C 180,E1 20578.764,E2 20578.764} C_VEL
LIN {X 0,Y 459.805,Z 723.341,A -85,B 0,C 180,E1 20577.364,E2 20577.364} C_VEL
LIN {X 0,Y 462.308,Z 703.547,A -85,B 0,C 180,E1 20576.18,E2 20576.18} C_VEL
LIN {X 0,Y 464.501,Z 682.09,A -85,B 0,C 180,E1 20575.144,E2 20575.144} C_VEL
LIN {X 0,Y 466.234,Z 659.826,A -85,B 0,C 180,E1 20574.319,E2 20574.319} C_VEL
LIN {X 0,Y 469.071,Z 618.252,A -85,B 0,C 180,E1 20573.169,E2 20573.169} C_VEL
LIN {X 0,Y 474.59,Z 546.788,A -85,B 0,C 180,E1 20571.525,E2 20571.525} C_VEL
LIN {X 0,Y 478.814,Z 480.116,A -85,B 0,C 180,E1 20570.21,E2 20570.21} C_VEL
LIN {X 0,Y 482.228,Z 404.363,A -85,B 0,C 180,E1 20568.963,E2 20568.963} C_VEL
LIN {X 0,Y 482.865,Z 388.766,A -85,B 0,C 180,E1 20568.716,E2 20568.716} C_VEL
LIN {X 0,Y 487.692,Z 367.209,A -85,B 0,C 180,E1 20567.9,E2 20567.9} C_VEL
LIN {X 0,Y 488.087,Z 337.279,A -85,B 0,C 180,E1 20565.808,E2 20565.808} C_VEL
LIN {X 0,Y 480.525,Z 316.786,A -85,B 0,C 180,E1 20563.204,E2 20563.204} C_VEL
LIN {X 0,Y 473.272,Z 299.429,A -85,B 0,C 180,E1 20560.756,E2 20560.756} C_VEL
LIN {X 0,Y 465.37,Z 283.001,A -85,B 0,C 180,E1 20558.228,E2 20558.228} C_VEL
LIN {X 0,Y 458.52,Z 270.201,A -85,B 0,C 180,E1 20556.071,E2 20556.071} C_VEL
LIN {X 0,Y 451.389,Z 257.758,A -85,B 0,C 180,E1 20553.78,E2 20553.78} C_VEL
LIN {X 0,Y 447.535,Z 251.832,A -85,B 0,C 180,E1 20552.578,E2 20552.578} C_VEL
LIN {X 0,Y 444.581,Z 247.118,A -85,B 0,C 180,E1 20551.603,E2 20551.603} C_VEL
LIN {X 0,Y 442.024,Z 242.9,A -85,B 0,C 180,E1 20550.73,E2 20550.73} C_VEL
LIN {X 0,Y 439.004,Z 238.993,A -85,B 0,C 180,E1 20549.77,E2 20549.77} C_VEL
LIN {X 0,Y 438.078,Z 236.858,A -85,B 0,C 180,E1 20549.389,E2 20549.389} C_VEL
LIN {X 0,Y 435.686,Z 234.524,A -85,B 0,C 180,E1 20548.663,E2 20548.663} C_VEL
LIN {X 0,Y 434.427,Z 231.152,A -85,B 0,C 180,E1 20548.082,E2 20548.082} C_VEL
LIN {X 0,Y 434.413,Z 231.077,A -85,B 0,C 180,E1 20544.186,E2 20544.186} C_VEL
LIN {X 0,Y 434.415,Z 231.111,A -85,B 0,C 180,E1 20540.479,E2 20540.479} C_VEL
LIN {X 0,Y 434.41,Z 231.082,A -85,B 0,C 180,E1 20536.721,E2 20536.721} C_VEL
LIN {X 0,Y 434.414,Z 231.07,A -85,B 0,C 180,E1 20533.036,E2 20533.036} C_VEL
LIN {X 0,Y 434.417,Z 231.117,A -85,B 0,C 180,E1 20529.138,E2 20529.138} C_VEL
LIN {X 0,Y 434.4,Z 231.067,A -85,B 0,C 180,E1 20525.415,E2 20525.415} C_VEL
LIN {X 0,Y 434.4,Z 231.102,A -85,B 0,C 180,E1 20521.583,E2 20521.583} C_VEL
LIN {X 0,Y 434.397,Z 231.086,A -85,B 0,C 180,E1 20517.757,E2 20517.757} C_VEL
LIN {X 0,Y 434.407,Z 231.074,A -85,B 0,C 180,E1 20514.055,E2 20514.055} C_VEL
LIN {X 0,Y 434.417,Z 231.109,A -85,B 0,C 180,E1 20510.327,E2 20510.327} C_VEL
LIN {X 0,Y 434.422,Z 231.116,A -85,B 0,C 180,E1 20506.558,E2 20506.558} C_VEL
LIN {X 0,Y 434.418,Z 231.119,A -85,B 0,C 180,E1 20502.727,E2 20502.727} C_VEL
LIN {X 0,Y 434.405,Z 231.11,A -85,B 0,C 180,E1 20498.957,E2 20498.957} C_VEL
LIN {X 0,Y 434.462,Z 231.349,A -85,B 0,C 180,E1 20498.393,E2 20498.393} C_VEL
LIN {X 0,Y 435.727,Z 234.638,A -85,B 0,C 180,E1 20497.751,E2 20497.751} C_VEL
LIN {X 0,Y 436.823,Z 236.057,A -85,B 0,C 180,E1 20497.384,E2 20497.384} C_VEL
LIN {X 0,Y 438.586,Z 239.757,A -85,B 0,C 180,E1 20496.629,E2 20496.629} C_VEL
LIN {X 0,Y 444.512,Z 251.087,A -85,B 0,C 180,E1 20494.27,E2 20494.27} C_VEL
LIN {X 0,Y 451.703,Z 264.954,A -85,B 0,C 180,E1 20491.58,E2 20491.58} C_VEL
LIN {X 0,Y 460.948,Z 283.156,A -85,B 0,C 180,E1 20488.335,E2 20488.335} C_VEL
LIN {X 0,Y 470.989,Z 303.713,A -85,B 0,C 180,E1 20485.026,E2 20485.026} C_VEL
LIN {X 0,Y 480.444,Z 323.416,A -85,B 0,C 180,E1 20482.181,E2 20482.181} C_VEL
LIN {X 0,Y 492.32,Z 342.331,A -85,B 0,C 180,E1 20480.538,E2 20480.538} C_VEL
LIN {X 0,Y 493.116,Z 353.729,A -85,B 0,C 180,E1 20480.189,E2 20480.189} C_VEL
LIN {X 0,Y 479.816,Z 597.99,A -85,B 0,C 180,E1 20475.783,E2 20475.783} C_VEL
LIN {X 0,Y 475.206,Z 693.32,A -85,B 0,C 180,E1 20474.055,E2 20474.055} C_VEL
LIN {X 0,Y 473.089,Z 717.844,A -85,B 0,C 180,E1 20473.411,E2 20473.411} C_VEL
LIN {X 0,Y 470.471,Z 742.347,A -85,B 0,C 180,E1 20472.561,E2 20472.561} C_VEL
LIN {X 0,Y 467.661,Z 764.279,A -85,B 0,C 180,E1 20471.596,E2 20471.596} C_VEL
LIN {X 0,Y 464.068,Z 788.83,A -85,B 0,C 180,E1 20470.27,E2 20470.27} C_VEL
LIN {X 0,Y 460.557,Z 810.563,A -85,B 0,C 180,E1 20468.861,E2 20468.861} C_VEL
LIN {X 0,Y 456.832,Z 831.454,A -85,B 0,C 180,E1 20467.242,E2 20467.242} C_VEL
LIN {X 0,Y 453.028,Z 851.892,A -85,B 0,C 180,E1 20465.403,E2 20465.403} C_VEL
LIN {X 0,Y 449.468,Z 870.25,A -85,B 0,C 180,E1 20463.464,E2 20463.464} C_VEL
LIN {X 0,Y 445.834,Z 888.842,A -85,B 0,C 180,E1 20461.203,E2 20461.203} C_VEL
LIN {X 0,Y 442.844,Z 904.158,A -85,B 0,C 180,E1 20459.042,E2 20459.042} C_VEL
LIN {X 0,Y 439.83,Z 920.376,A -85,B 0,C 180,E1 20456.401,E2 20456.401} C_VEL
LIN {X 0,Y 437.547,Z 933.458,A -85,B 0,C 180,E1 20453.923,E2 20453.923} C_VEL
LIN {X 0,Y 435.492,Z 946.713,A -85,B 0,C 180,E1 20450.988,E2 20450.988} C_VEL
LIN {X 0,Y 434.204,Z 956.661,A -85,B 0,C 180,E1 20448.39,E2 20448.39} C_VEL
LIN {X 0,Y 433.18,Z 966.726,A -85,B 0,C 180,E1 20445.235,E2 20445.235} C_VEL
LIN {X 0,Y 432.709,Z 973.704,A -85,B 0,C 180,E1 20442.545,E2 20442.545} C_VEL
LIN {X 0,Y 432.51,Z 980.015,A -85,B 0,C 180,E1 20439.447,E2 20439.447} C_VEL
LIN {X 0,Y 432.525,Z 983.969,A -85,B 0,C 180,E1 20436.771,E2 20436.771} C_VEL
LIN {X 0,Y 432.609,Z 986.642,A -85,B 0,C 180,E1 20434.109,E2 20434.109} C_VEL
LIN {X 0,Y 432.684,Z 988.026,A -85,B 0,C 180,E1 20431.059,E2 20431.059} C_VEL
LIN {X 0,Y 432.693,Z 987.865,A -85,B 0,C 180,E1 20428.543,E2 20428.543} C_VEL
LIN {X 0,Y 432.625,Z 986.465,A -85,B 0,C 180,E1 20425.891,E2 20425.891} C_VEL
LIN {X 0,Y 432.518,Z 983.402,A -85,B 0,C 180,E1 20422.962,E2 20422.962} C_VEL
LIN {X 0,Y 432.535,Z 978.948,A -85,B 0,C 180,E1 20420.15,E2 20420.15} C_VEL
LIN {X 0,Y 432.746,Z 972.775,A -85,B 0,C 180,E1 20417.178,E2 20417.178} C_VEL
LIN {X 0,Y 433.299,Z 964.787,A -85,B 0,C 180,E1 20414.199,E2 20414.199} C_VEL
LIN {X 0,Y 434.282,Z 955.593,A -85,B 0,C 180,E1 20411.335,E2 20411.335} C_VEL
LIN {X 0,Y 435.918,Z 943.785,A -85,B 0,C 180,E1 20408.276,E2 20408.276} C_VEL
LIN {X 0,Y 438.19,Z 930.428,A -85,B 0,C 180,E1 20405.318,E2 20405.318} C_VEL
LIN {X 0,Y 440.937,Z 915.903,A -85,B 0,C 180,E1 20402.591,E2 20402.591} C_VEL
LIN {X 0,Y 444.43,Z 899.316,A -85,B 0,C 180,E1 20399.887,E2 20399.887} C_VEL
LIN {X 0,Y 447.961,Z 883.142,A -85,B 0,C 180,E1 20397.608,E2 20397.608} C_VEL
LIN {X 0,Y 452.503,Z 863.23,A -85,B 0,C 180,E1 20395.174,E2 20395.174} C_VEL
LIN {X 0,Y 457.214,Z 842.793,A -85,B 0,C 180,E1 20393.029,E2 20393.029} C_VEL
LIN {X 0,Y 461.973,Z 821.362,A -85,B 0,C 180,E1 20391.121,E2 20391.121} C_VEL
LIN {X 0,Y 466.951,Z 798.439,A -85,B 0,C 180,E1 20389.386,E2 20389.386} C_VEL
LIN {X 0,Y 471.451,Z 776.7,A -85,B 0,C 180,E1 20387.999,E2 20387.999} C_VEL
LIN {X 0,Y 475.647,Z 754.482,A -85,B 0,C 180,E1 20386.823,E2 20386.823} C_VEL
LIN {X 0,Y 479.769,Z 730.807,A -85,B 0,C 180,E1 20385.794,E2 20385.794} C_VEL
LIN {X 0,Y 483.218,Z 708.005,A -85,B 0,C 180,E1 20385.011,E2 20385.011} C_VEL
LIN {X 0,Y 486.34,Z 682.731,A -85,B 0,C 180,E1 20384.352,E2 20384.352} C_VEL
LIN {X 0,Y 494.076,Z 612.481,A -85,B 0,C 180,E1 20382.794,E2 20382.794} C_VEL
LIN {X 0,Y 502.506,Z 553.906,A -85,B 0,C 180,E1 20381.417,E2 20381.417} C_VEL
LIN {X 0,Y 513.155,Z 495.233,A -85,B 0,C 180,E1 20379.987,E2 20379.987} C_VEL
LIN {X 0,Y 520.231,Z 462.048,A -85,B 0,C 180,E1 20379.17,E2 20379.17} C_VEL
LIN {X 0,Y 514.117,Z 487.384,A -85,B 0,C 180,E1 20377.631,E2 20377.631} C_VEL
LIN {X 0,Y 508.478,Z 516.377,A -85,B 0,C 180,E1 20376.083,E2 20376.083} C_VEL
LIN {X 0,Y 507.364,Z 522.401,A -85,B 0,C 180,E1 20375.825,E2 20375.825} C_VEL
LIN {X 0,Y 487.121,Z 627.358,A -85,B 0,C 180,E1 20372.743,E2 20372.743} C_VEL
LIN {X 0,Y 475.859,Z 693.759,A -85,B 0,C 180,E1 20370.651,E2 20370.651} C_VEL
LIN {X 0,Y 471.445,Z 717.142,A -85,B 0,C 180,E1 20369.685,E2 20369.685} C_VEL
LIN {X 0,Y 466.821,Z 740.453,A -85,B 0,C 180,E1 20368.462,E2 20368.462} C_VEL
LIN {X 0,Y 462.255,Z 762.889,A -85,B 0,C 180,E1 20367.017,E2 20367.017} C_VEL
LIN {X 0,Y 457.972,Z 783.621,A -85,B 0,C 180,E1 20365.405,E2 20365.405} C_VEL
LIN {X 0,Y 454.035,Z 802.687,A -85,B 0,C 180,E1 20363.629,E2 20363.629} C_VEL
LIN {X 0,Y 450.491,Z 819.554,A -85,B 0,C 180,E1 20361.757,E2 20361.757} C_VEL
LIN {X 0,Y 447.216,Z 834.742,A -85,B 0,C 180,E1 20359.731,E2 20359.731} C_VEL
LIN {X 0,Y 444.24,Z 848.199,A -85,B 0,C 180,E1 20357.554,E2 20357.554} C_VEL
LIN {X 0,Y 441.869,Z 858.654,A -85,B 0,C 180,E1 20355.487,E2 20355.487} C_VEL
LIN {X 0,Y 439.826,Z 867.472,A -85,B 0,C 180,E1 20353.343,E2 20353.343} C_VEL
LIN {X 0,Y 437.956,Z 875.128,A -85,B 0,C 180,E1 20350.923,E2 20350.923} C_VEL
LIN {X 0,Y 436.551,Z 880.519,A -85,B 0,C 180,E1 20348.562,E2 20348.562} C_VEL
LIN {X 0,Y 435.506,Z 884.037,A -85,B 0,C 180,E1 20346.195,E2 20346.195} C_VEL
LIN {X 0,Y 434.739,Z 885.709,A -85,B 0,C 180,E1 20343.824,E2 20343.824} C_VEL
LIN {X 0,Y 434.252,Z 885.662,A -85,B 0,C 180,E1 20341.583,E2 20341.583} C_VEL
LIN {X 0,Y 433.949,Z 883.916,A -85,B 0,C 180,E1 20339.208,E2 20339.208} C_VEL
LIN {X 0,Y 433.822,Z 880.414,A -85,B 0,C 180,E1 20336.829,E2 20336.829} C_VEL
LIN {X 0,Y 433.898,Z 875.128,A -85,B 0,C 180,E1 20334.446,E2 20334.446} C_VEL
LIN {X 0,Y 434.191,Z 867.946,A -85,B 0,C 180,E1 20332.058,E2 20332.058} C_VEL
LIN {X 0,Y 434.752,Z 858.696,A -85,B 0,C 180,E1 20329.666,E2 20329.666} C_VEL
LIN {X 0,Y 435.588,Z 847.848,A -85,B 0,C 180,E1 20327.404,E2 20327.404} C_VEL
LIN {X 0,Y 436.677,Z 835.492,A -85,B 0,C 180,E1 20325.276,E2 20325.276} C_VEL
LIN {X 0,Y 438.002,Z 821.663,A -85,B 0,C 180,E1 20323.283,E2 20323.283} C_VEL
LIN {X 0,Y 439.526,Z 806.355,A -85,B 0,C 180,E1 20321.428,E2 20321.428} C_VEL
LIN {X 0,Y 441.297,Z 788.852,A -85,B 0,C 180,E1 20319.647,E2 20319.647} C_VEL
LIN {X 0,Y 443.116,Z 770.098,A -85,B 0,C 180,E1 20318.064,E2 20318.064} C_VEL
LIN {X 0,Y 444.956,Z 750.504,A -85,B 0,C 180,E1 20316.703,E2 20316.703} C_VEL
LIN {X 0,Y 446.74,Z 729.864,A -85,B 0,C 180,E1 20315.539,E2 20315.539} C_VEL
LIN {X 0,Y 448.439,Z 707.503,A -85,B 0,C 180,E1 20314.552,E2 20314.552} C_VEL
LIN {X 0,Y 449.902,Z 685.211,A -85,B 0,C 180,E1 20313.822,E2 20313.822} C_VEL
LIN {X 0,Y 458.982,Z 504.432,A -85,B 0,C 180,E1 20309.816,E2 20309.816} C_VEL
LIN {X 0,Y 453.98,Z 440.307,A -85,B 0,C 180,E1 20307.791,E2 20307.791} C_VEL
LIN {X 0,Y 459.668,Z 389.317,A -85,B 0,C 180,E1 20303.724,E2 20303.724} C_VEL
LIN {X 0,Y 465.95,Z 337.928,A -85,B 0,C 180,E1 20299.604,E2 20299.604} C_VEL
LIN {X 0,Y 468.304,Z 320.279,A -85,B 0,C 180,E1 20298.187,E2 20298.187} C_VEL
LIN {X 0,Y 469.999,Z 320.421,A -85,B 0,C 180,E1 20297.922,E2 20297.922} C_VEL
LIN {X 0,Y 472.95,Z 319.101,A -85,B 0,C 180,E1 20297.591,E2 20297.591} C_VEL
LIN {X 0,Y 473.758,Z 318.551,A -85,B 0,C 180,E1 20297.516,E2 20297.516} C_VEL
LIN {X 0,Y 481.12,Z 318.541,A -85,B 0,C 180,E1 20296.453,E2 20296.453} C_VEL
LIN {X 0,Y 488.11,Z 337.655,A -85,B 0,C 180,E1 20294.047,E2 20294.047} C_VEL
LIN {X 0,Y 487.583,Z 367.186,A -85,B 0,C 180,E1 20291.997,E2 20291.997} C_VEL
LIN {X 0,Y 482.724,Z 389.848,A -85,B 0,C 180,E1 20291.164,E2 20291.164} C_VEL
LIN {X 0,Y 479.12,Z 473.033,A -85,B 0,C 180,E1 20289.817,E2 20289.817} C_VEL
LIN {X 0,Y 475.182,Z 537.396,A -85,B 0,C 180,E1 20288.573,E2 20288.573} C_VEL
LIN {X 0,Y 469.914,Z 606.927,A -85,B 0,C 180,E1 20287.007,E2 20287.007} C_VEL
LIN {X 0,Y 466.667,Z 651.872,A -85,B 0,C 180,E1 20285.827,E2 20285.827} C_VEL
LIN {X 0,Y 465.17,Z 673.986,A -85,B 0,C 180,E1 20285.085,E2 20285.085} C_VEL
LIN {X 0,Y 463.302,Z 694.051,A -85,B 0,C 180,E1 20284.209,E2 20284.209} C_VEL
LIN {X 0,Y 463.124,Z 695.785,A -85,B 0,C 180,E1 20284.124,E2 20284.124} C_VEL
LIN {X 0,Y 461.533,Z 703.006,A -85,B 0,C 180,E1 20283.829,E2 20283.829} C_VEL
LIN {X 0,Y 454.331,Z 721.147,A -85,B 0,C 180,E1 20283.208,E2 20283.208} C_VEL
LIN {X 0,Y 452.526,Z 727.999,A -85,B 0,C 180,E1 20282.82,E2 20282.82} C_VEL
LIN {X 0,Y 449.433,Z 747.73,A -85,B 0,C 180,E1 20281.315,E2 20281.315} C_VEL
LIN {X 0,Y 446.115,Z 766.61,A -85,B 0,C 180,E1 20279.583,E2 20279.583} C_VEL
LIN {X 0,Y 442.734,Z 784.281,A -85,B 0,C 180,E1 20277.653,E2 20277.653} C_VEL
LIN {X 0,Y 439.536,Z 800.082,A -85,B 0,C 180,E1 20275.609,E2 20275.609} C_VEL
LIN {X 0,Y 436.629,Z 814.087,A -85,B 0,C 180,E1 20273.482,E2 20273.482} C_VEL
LIN {X 0,Y 433.818,Z 827.523,A -85,B 0,C 180,E1 20271.073,E2 20271.073} C_VEL
LIN {X 0,Y 431.257,Z 840.011,A -85,B 0,C 180,E1 20268.38,E2 20268.38} C_VEL
LIN {X 0,Y 429.163,Z 850.783,A -85,B 0,C 180,E1 20265.541,E2 20265.541} C_VEL
LIN {X 0,Y 427.642,Z 859.422,A -85,B 0,C 180,E1 20262.697,E2 20262.697} C_VEL
LIN {X 0,Y 426.613,Z 865.849,A -85,B 0,C 180,E1 20259.988,E2 20259.988} C_VEL
LIN {X 0,Y 425.948,Z 870.878,A -85,B 0,C 180,E1 20257.147,E2 20257.147} C_VEL
LIN {X 0,Y 425.573,Z 874.236,A -85,B 0,C 180,E1 20254.312,E2 20254.312} C_VEL
LIN {X 0,Y 425.411,Z 875.978,A -85,B 0,C 180,E1 20251.482,E2 20251.482} C_VEL
LIN {X 0,Y 425.396,Z 876.037,A -85,B 0,C 180,E1 20248.788,E2 20248.788} C_VEL
LIN {X 0,Y 425.541,Z 874.534,A -85,B 0,C 180,E1 20245.958,E2 20245.958} C_VEL
LIN {X 0,Y 425.89,Z 871.42,A -85,B 0,C 180,E1 20243.123,E2 20243.123} C_VEL
LIN {X 0,Y 426.517,Z 866.643,A -85,B 0,C 180,E1 20240.283,E2 20240.283} C_VEL
LIN {X 0,Y 427.548,Z 860.065,A -85,B 0,C 180,E1 20237.438,E2 20237.438} C_VEL
LIN {X 0,Y 429.023,Z 851.551,A -85,B 0,C 180,E1 20234.592,E2 20234.592} C_VEL
LIN {X 0,Y 430.845,Z 842.034,A -85,B 0,C 180,E1 20232.021,E2 20232.021} C_VEL
LIN {X 0,Y 433.169,Z 830.622,A -85,B 0,C 180,E1 20229.46,E2 20229.46} C_VEL
LIN {X 0,Y 436.027,Z 817.006,A -85,B 0,C 180,E1 20226.913,E2 20226.913} C_VEL
LIN {X 0,Y 439.047,Z 802.603,A -85,B 0,C 180,E1 20224.65,E2 20224.65} C_VEL
LIN {X 0,Y 442.22,Z 787.088,A -85,B 0,C 180,E1 20222.583,E2 20222.583} C_VEL
LIN {X 0,Y 445.46,Z 770.482,A -85,B 0,C 180,E1 20220.704,E2 20220.704} C_VEL
LIN {X 0,Y 448.778,Z 752.101,A -85,B 0,C 180,E1 20218.95,E2 20218.95} C_VEL
LIN {X 0,Y 451.954,Z 732.415,A -85,B 0,C 180,E1 20217.384,E2 20217.384} C_VEL
LIN {X 0,Y 454.795,Z 712.053,A -85,B 0,C 180,E1 20216.053,E2 20216.053} C_VEL
LIN {X 0,Y 457.165,Z 691.454,A -85,B 0,C 180,E1 20214.961,E2 20214.961} C_VEL
LIN {X 0,Y 459.051,Z 670.445,A -85,B 0,C 180,E1 20214.083,E2 20214.083} C_VEL
LIN {X 0,Y 460.847,Z 643.521,A -85,B 0,C 180,E1 20213.238,E2 20213.238} C_VEL
LIN {X 0,Y 465.018,Z 591.098,A -85,B 0,C 180,E1 20211.899,E2 20211.899} C_VEL
LIN {X 0,Y 469.955,Z 525.918,A -85,B 0,C 180,E1 20210.459,E2 20210.459} C_VEL
LIN {X 0,Y 473.829,Z 460.766,A -85,B 0,C 180,E1 20209.231,E2 20209.231} C_VEL
LIN {X 0,Y 476.944,Z 390.939,A -85,B 0,C 180,E1 20208.094,E2 20208.094} C_VEL
LIN {X 0,Y 481.922,Z 368.425,A -85,B 0,C 180,E1 20207.236,E2 20207.236} C_VEL
LIN {X 0,Y 482.284,Z 341.272,A -85,B 0,C 180,E1 20205.327,E2 20205.327} C_VEL
LIN {X 0,Y 474.795,Z 320.884,A -85,B 0,C 180,E1 20202.697,E2 20202.697} C_VEL
LIN {X 0,Y 467.967,Z 304.452,A -85,B 0,C 180,E1 20200.347,E2 20200.347} C_VEL
LIN {X 0,Y 459.483,Z 286.611,A -85,B 0,C 180,E1 20197.54,E2 20197.54} C_VEL
LIN {X 0,Y 451.665,Z 272.099,A -85,B 0,C 180,E1 20194.986,E2 20194.986} C_VEL
LIN {X 0,Y 444.206,Z 259.342,A -85,B 0,C 180,E1 20192.546,E2 20192.546} C_VEL
LIN {X 0,Y 440.149,Z 253.195,A -85,B 0,C 180,E1 20191.195,E2 20191.195} C_VEL
LIN {X 0,Y 437.232,Z 248.646,A -85,B 0,C 180,E1 20190.206,E2 20190.206} C_VEL
LIN {X 0,Y 434.72,Z 244.895,A -85,B 0,C 180,E1 20189.335,E2 20189.335} C_VEL
LIN {X 0,Y 434.076,Z 243.594,A -85,B 0,C 180,E1 20189.081,E2 20189.081} C_VEL
LIN {X 0,Y 431.481,Z 240.519,A -85,B 0,C 180,E1 20188.212,E2 20188.212} C_VEL
LIN {X 0,Y 430.122,Z 237.835,A -85,B 0,C 180,E1 20187.663,E2 20187.663} C_VEL
LIN {X 0,Y 427.62,Z 235.33,A -85,B 0,C 180,E1 20186.826,E2 20186.826} C_VEL
LIN {X 0,Y 426.48,Z 232.123,A -85,B 0,C 180,E1 20186.261,E2 20186.261} C_VEL
LIN {X 0,Y 426.481,Z 232.07,A -85,B 0,C 180,E1 20182.322,E2 20182.322} C_VEL
LIN {X 0,Y 426.472,Z 232.056,A -85,B 0,C 180,E1 20178.452,E2 20178.452} C_VEL
LIN {X 0,Y 426.474,Z 232.097,A -85,B 0,C 180,E1 20174.668,E2 20174.668} C_VEL
LIN {X 0,Y 426.473,Z 232.069,A -85,B 0,C 180,E1 20170.775,E2 20170.775} C_VEL
LIN {X 0,Y 426.483,Z 232.059,A -85,B 0,C 180,E1 20167.003,E2 20167.003} C_VEL
LIN {X 0,Y 426.472,Z 232.107,A -85,B 0,C 180,E1 20163.091,E2 20163.091} C_VEL
LIN {X 0,Y 426.46,Z 232.051,A -85,B 0,C 180,E1 20159.328,E2 20159.328} C_VEL
LIN {X 0,Y 426.46,Z 232.102,A -85,B 0,C 180,E1 20155.428,E2 20155.428} C_VEL
LIN {X 0,Y 426.452,Z 232.062,A -85,B 0,C 180,E1 20151.641,E2 20151.641} C_VEL
LIN {X 0,Y 426.462,Z 232.111,A -85,B 0,C 180,E1 20147.818,E2 20147.818} C_VEL
LIN {X 0,Y 426.468,Z 232.097,A -85,B 0,C 180,E1 20144.004,E2 20144.004} C_VEL
LIN {X 0,Y 426.476,Z 232.108,A -85,B 0,C 180,E1 20140.126,E2 20140.126} C_VEL
LIN {X 0,Y 426.478,Z 232.265,A -85,B 0,C 180,E1 20139.728,E2 20139.728} C_VEL
LIN {X 0,Y 427.763,Z 235.579,A -85,B 0,C 180,E1 20139.045,E2 20139.045} C_VEL
LIN {X 0,Y 429.097,Z 237.552,A -85,B 0,C 180,E1 20138.54,E2 20138.54} C_VEL
LIN {X 0,Y 430.846,Z 241.073,A -85,B 0,C 180,E1 20137.772,E2 20137.772} C_VEL
LIN {X 0,Y 436.457,Z 251.678,A -85,B 0,C 180,E1 20135.502,E2 20135.502} C_VEL
LIN {X 0,Y 443.835,Z 266.001,A -85,B 0,C 180,E1 20132.64,E2 20132.64} C_VEL
LIN {X 0,Y 452.566,Z 283.268,A -85,B 0,C 180,E1 20129.459,E2 20129.459} C_VEL
LIN {X 0,Y 462.107,Z 302.657,A -85,B 0,C 180,E1 20126.214,E2 20126.214} C_VEL
LIN {X 0,Y 472.195,Z 323.815,A -85,B 0,C 180,E1 20123.031,E2 20123.031} C_VEL
LIN {X 0,Y 486.355,Z 346.135,A -85,B 0,C 180,E1 20121.035,E2 20121.035} C_VEL
LIN {X 0,Y 486.887,Z 355.043,A -85,B 0,C 180,E1 20120.765,E2 20120.765} C_VEL
LIN {X 0,Y 473.101,Z 598.027,A -85,B 0,C 180,E1 20116.306,E2 20116.306} C_VEL
LIN {X 0,Y 468.309,Z 693.219,A -85,B 0,C 180,E1 20114.549,E2 20114.549} C_VEL
LIN {X 0,Y 466.145,Z 717.602,A -85,B 0,C 180,E1 20113.899,E2 20113.899} C_VEL
LIN {X 0,Y 463.515,Z 741.606,A -85,B 0,C 180,E1 20113.059,E2 20113.059} C_VEL
LIN {X 0,Y 460.717,Z 762.87,A -85,B 0,C 180,E1 20112.115,E2 20112.115} C_VEL
LIN {X 0,Y 457.151,Z 786.865,A -85,B 0,C 180,E1 20110.819,E2 20110.819} C_VEL
LIN {X 0,Y 453.657,Z 807.865,A -85,B 0,C 180,E1 20109.452,E2 20109.452} C_VEL
LIN {X 0,Y 449.741,Z 829.66,A -85,B 0,C 180,E1 20107.771,E2 20107.771} C_VEL
LIN {X 0,Y 445.89,Z 849.884,A -85,B 0,C 180,E1 20105.95,E2 20105.95} C_VEL
LIN {X 0,Y 442.14,Z 868.681,A -85,B 0,C 180,E1 20103.958,E2 20103.958} C_VEL
LIN {X 0,Y 438.483,Z 886.955,A -85,B 0,C 180,E1 20101.726,E2 20101.726} C_VEL
LIN {X 0,Y 435.26,Z 902.953,A -85,B 0,C 180,E1 20099.446,E2 20099.446} C_VEL
LIN {X 0,Y 432.19,Z 918.993,A -85,B 0,C 180,E1 20096.817,E2 20096.817} C_VEL
LIN {X 0,Y 429.947,Z 931.377,A -85,B 0,C 180,E1 20094.454,E2 20094.454} C_VEL
LIN {X 0,Y 427.893,Z 944.08,A -85,B 0,C 180,E1 20091.667,E2 20091.667} C_VEL
LIN {X 0,Y 426.398,Z 954.751,A -85,B 0,C 180,E1 20088.881,E2 20088.881} C_VEL
LIN {X 0,Y 425.364,Z 964.265,A -85,B 0,C 180,E1 20085.964,E2 20085.964} C_VEL
LIN {X 0,Y 424.793,Z 972.078,A -85,B 0,C 180,E1 20082.969,E2 20082.969} C_VEL
LIN {X 0,Y 424.553,Z 978.232,A -85,B 0,C 180,E1 20080.037,E2 20080.037} C_VEL
LIN {X 0,Y 424.551,Z 982.756,A -85,B 0,C 180,E1 20077.035,E2 20077.035} C_VEL
LIN {X 0,Y 424.647,Z 985.404,A -85,B 0,C 180,E1 20074.456,E2 20074.456} C_VEL
LIN {X 0,Y 424.735,Z 987.033,A -85,B 0,C 180,E1 20071.484,E2 20071.484} C_VEL
LIN {X 0,Y 424.748,Z 986.967,A -85,B 0,C 180,E1 20068.651,E2 20068.651} C_VEL
LIN {X 0,Y 424.675,Z 985.626,A -85,B 0,C 180,E1 20065.949,E2 20065.949} C_VEL
LIN {X 0,Y 424.549,Z 982.683,A -85,B 0,C 180,E1 20062.965,E2 20062.965} C_VEL
LIN {X 0,Y 424.556,Z 978.274,A -85,B 0,C 180,E1 20060.1,E2 20060.1} C_VEL
LIN {X 0,Y 424.75,Z 972.469,A -85,B 0,C 180,E1 20057.216,E2 20057.216} C_VEL
LIN {X 0,Y 425.336,Z 964.289,A -85,B 0,C 180,E1 20054.035,E2 20054.035} C_VEL
LIN {X 0,Y 426.303,Z 955.621,A -85,B 0,C 180,E1 20051.256,E2 20051.256} C_VEL
LIN {X 0,Y 428.057,Z 943.596,A -85,B 0,C 180,E1 20048.025,E2 20048.025} C_VEL
LIN {X 0,Y 430.2,Z 931.534,A -85,B 0,C 180,E1 20045.269,E2 20045.269} C_VEL
LIN {X 0,Y 433.18,Z 916.69,A -85,B 0,C 180,E1 20042.357,E2 20042.357} C_VEL
LIN {X 0,Y 436.804,Z 900.467,A -85,B 0,C 180,E1 20039.609,E2 20039.609} C_VEL
LIN {X 0,Y 440.698,Z 883.603,A -85,B 0,C 180,E1 20037.162,E2 20037.162} C_VEL
LIN {X 0,Y 445.139,Z 865.398,A -85,B 0,C 180,E1 20034.849,E2 20034.849} C_VEL
LIN {X 0,Y 449.915,Z 845.746,A -85,B 0,C 180,E1 20032.714,E2 20032.714} C_VEL
LIN {X 0,Y 455.25,Z 823.443,A -85,B 0,C 180,E1 20030.635,E2 20030.635} C_VEL
LIN {X 0,Y 460.376,Z 801.638,A -85,B 0,C 180,E1 20028.908,E2 20028.908} C_VEL
LIN {X 0,Y 465.154,Z 780.008,A -85,B 0,C 180,E1 20027.475,E2 20027.475} C_VEL
LIN {X 0,Y 470.242,Z 755.462,A -85,B 0,C 180,E1 20026.117,E2 20026.117} C_VEL
LIN {X 0,Y 474.678,Z 732.122,A -85,B 0,C 180,E1 20025.07,E2 20025.07} C_VEL
LIN {X 0,Y 478.408,Z 709.551,A -85,B 0,C 180,E1 20024.269,E2 20024.269} C_VEL
LIN {X 0,Y 482.08,Z 683.101,A -85,B 0,C 180,E1 20023.55,E2 20023.55} C_VEL
LIN {X 0,Y 490.399,Z 615.868,A -85,B 0,C 180,E1 20022.012,E2 20022.012} C_VEL
LIN {X 0,Y 499.619,Z 558.231,A -85,B 0,C 180,E1 20020.63,E2 20020.63} C_VEL
LIN {X 0,Y 510.732,Z 502.233,A -85,B 0,C 180,E1 20019.253,E2 20019.253} C_VEL
LIN {X 0,Y 514.736,Z 484.385,A -85,B 0,C 180,E1 20018.799,E2 20018.799} C_VEL
LIN {X 0,Y 508.019,Z 513.092,A -85,B 0,C 180,E1 20017.219,E2 20017.219} C_VEL
LIN {X 0,Y 505.729,Z 524.168,A -85,B 0,C 180,E1 20016.689,E2 20016.689} C_VEL
LIN {X 0,Y 484.235,Z 628.309,A -85,B 0,C 180,E1 20013.618,E2 20013.618} C_VEL
LIN {X 0,Y 472.206,Z 693.862,A -85,B 0,C 180,E1 20011.526,E2 20011.526} C_VEL
LIN {X 0,Y 467.335,Z 717.432,A -85,B 0,C 180,E1 20010.541,E2 20010.541} C_VEL
LIN {X 0,Y 462.141,Z 741.15,A -85,B 0,C 180,E1 20009.273,E2 20009.273} C_VEL
LIN {X 0,Y 457.024,Z 763.873,A -85,B 0,C 180,E1 20007.776,E2 20007.776} C_VEL
LIN {X 0,Y 452.238,Z 784.865,A -85,B 0,C 180,E1 20006.103,E2 20006.103} C_VEL
LIN {X 0,Y 447.854,Z 804.185,A -85,B 0,C 180,E1 20004.255,E2 20004.255} C_VEL
LIN {X 0,Y 443.79,Z 821.736,A -85,B 0,C 180,E1 20002.242,E2 20002.242} C_VEL
LIN {X 0,Y 440.509,Z 835.783,A -85,B 0,C 180,E1 20000.322,E2 20000.322} C_VEL
LIN {X 0,Y 437.482,Z 848.495,A -85,B 0,C 180,E1 19998.248,E2 19998.248} C_VEL
LIN {X 0,Y 434.746,Z 859.667,A -85,B 0,C 180,E1 19996.021,E2 19996.021} C_VEL
LIN {X 0,Y 432.329,Z 869.151,A -85,B 0,C 180,E1 19993.645,E2 19993.645} C_VEL
LIN {X 0,Y 430.476,Z 876.136,A -85,B 0,C 180,E1 19991.387,E2 19991.387} C_VEL
LIN {X 0,Y 428.936,Z 881.586,A -85,B 0,C 180,E1 19988.985,E2 19988.985} C_VEL
LIN {X 0,Y 427.775,Z 885.109,A -85,B 0,C 180,E1 19986.577,E2 19986.577} C_VEL
LIN {X 0,Y 426.964,Z 886.798,A -85,B 0,C 180,E1 19984.298,E2 19984.298} C_VEL
LIN {X 0,Y 426.376,Z 886.86,A -85,B 0,C 180,E1 19981.881,E2 19981.881} C_VEL
LIN {X 0,Y 426.029,Z 885.173,A -85,B 0,C 180,E1 19979.462,E2 19979.462} C_VEL
LIN {X 0,Y 425.876,Z 881.732,A -85,B 0,C 180,E1 19977.039,E2 19977.039} C_VEL
LIN {X 0,Y 425.933,Z 876.496,A -85,B 0,C 180,E1 19974.612,E2 19974.612} C_VEL
LIN {X 0,Y 426.194,Z 869.835,A -85,B 0,C 180,E1 19972.315,E2 19972.315} C_VEL
LIN {X 0,Y 426.693,Z 861.334,A -85,B 0,C 180,E1 19970.014,E2 19970.014} C_VEL
LIN {X 0,Y 427.493,Z 850.799,A -85,B 0,C 180,E1 19967.711,E2 19967.711} C_VEL
LIN {X 0,Y 428.563,Z 838.672,A -85,B 0,C 180,E1 19965.523,E2 19965.523} C_VEL
LIN {X 0,Y 429.957,Z 824.273,A -85,B 0,C 180,E1 19963.362,E2 19963.362} C_VEL
LIN {X 0,Y 431.592,Z 808.256,A -85,B 0,C 180,E1 19961.354,E2 19961.354} C_VEL
LIN {X 0,Y 433.399,Z 790.898,A -85,B 0,C 180,E1 19959.535,E2 19959.535} C_VEL
LIN {X 0,Y 435.327,Z 771.859,A -85,B 0,C 180,E1 19957.871,E2 19957.871} C_VEL
LIN {X 0,Y 437.202,Z 752.517,A -85,B 0,C 180,E1 19956.486,E2 19956.486} C_VEL
LIN {X 0,Y 439.035,Z 732.107,A -85,B 0,C 180,E1 19955.297,E2 19955.297} C_VEL
LIN {X 0,Y 440.764,Z 710.262,A -85,B 0,C 180,E1 19954.292,E2 19954.292} C_VEL
LIN {X 0,Y 442.336,Z 687.29,A -85,B 0,C 180,E1 19953.502,E2 19953.502} C_VEL
LIN {X 0,Y 444.209,Z 649.813,A -85,B 0,C 180,E1 19952.615,E2 19952.615} C_VEL
LIN {X 0,Y 451.822,Z 505.136,A -85,B 0,C 180,E1 19949.367,E2 19949.367} C_VEL
LIN {X 0,Y 446.865,Z 439.5,A -85,B 0,C 180,E1 19947.249,E2 19947.249} C_VEL
LIN {X 0,Y 452.749,Z 388.876,A -85,B 0,C 180,E1 19943.158,E2 19943.158} C_VEL
LIN {X 0,Y 459.417,Z 336.523,A -85,B 0,C 180,E1 19938.907,E2 19938.907} C_VEL
LIN {X 0,Y 460.11,Z 332.118,A -85,B 0,C 180,E1 19938.531,E2 19938.531} C_VEL
LIN {X 0,Y 462.16,Z 332.055,A -85,B 0,C 180,E1 19938.213,E2 19938.213} C_VEL
LIN {X 0,Y 465.142,Z 330.415,A -85,B 0,C 180,E1 19937.879,E2 19937.879} C_VEL
LIN {X 0,Y 468.433,Z 327.76,A -85,B 0,C 180,E1 19937.583,E2 19937.583} C_VEL
LIN {X 0,Y 473.439,Z 325.91,A -85,B 0,C 180,E1 19936.986,E2 19936.986} C_VEL
LIN {X 0,Y 476.656,Z 325.887,A -85,B 0,C 180,E1 19936.524,E2 19936.524} C_VEL
LIN {X 0,Y 482.321,Z 341.882,A -85,B 0,C 180,E1 19934.509,E2 19934.509} C_VEL
LIN {X 0,Y 481.738,Z 369.053,A -85,B 0,C 180,E1 19932.626,E2 19932.626} C_VEL
LIN {X 0,Y 476.687,Z 392.56,A -85,B 0,C 180,E1 19931.765,E2 19931.765} C_VEL
LIN {X 0,Y 472.973,Z 475.5,A -85,B 0,C 180,E1 19930.41,E2 19930.41} C_VEL
LIN {X 0,Y 468.98,Z 538.697,A -85,B 0,C 180,E1 19929.175,E2 19929.175} C_VEL
LIN {X 0,Y 463.668,Z 606.761,A -85,B 0,C 180,E1 19927.625,E2 19927.625} C_VEL
LIN {X 0,Y 460.239,Z 651.951,A -85,B 0,C 180,E1 19926.421,E2 19926.421} C_VEL
LIN {X 0,Y 458.656,Z 674.727,A -85,B 0,C 180,E1 19925.654,E2 19925.654} C_VEL
LIN {X 0,Y 456.595,Z 696.121,A -85,B 0,C 180,E1 19924.706,E2 19924.706} C_VEL
LIN {X 0,Y 454.077,Z 716.813,A -85,B 0,C 180,E1 19923.553,E2 19923.553} C_VEL
LIN {X 0,Y 452.526,Z 727.999,A -85,B 0,C 180,E1 19922.82,E2 19922.82} C_VEL
LIN {X 0,Y 450.699,Z 734.854,A -85,B 0,C 180,E1 19922.408,E2 19922.408} C_VEL
LIN {X 0,Y 442.928,Z 751.978,A -85,B 0,C 180,E1 19921.493,E2 19921.493} C_VEL
LIN {X 0,Y 440.936,Z 758.361,A -85,B 0,C 180,E1 19920.992,E2 19920.992} C_VEL
LIN {X 0,Y 437.431,Z 776.665,A -85,B 0,C 180,E1 19919.136,E2 19919.136} C_VEL
LIN {X 0,Y 433.922,Z 793.74,A -85,B 0,C 180,E1 19917.072,E2 19917.072} C_VEL
LIN {X 0,Y 430.589,Z 809.209,A -85,B 0,C 180,E1 19914.854,E2 19914.854} C_VEL
LIN {X 0,Y 427.587,Z 822.933,A -85,B 0,C 180,E1 19912.528,E2 19912.528} C_VEL
LIN {X 0,Y 424.814,Z 835.676,A -85,B 0,C 180,E1 19909.955,E2 19909.955} C_VEL
LIN {X 0,Y 422.444,Z 846.943,A -85,B 0,C 180,E1 19907.21,E2 19907.21} C_VEL
LIN {X 0,Y 420.551,Z 856.578,A -85,B 0,C 180,E1 19904.316,E2 19904.316} C_VEL
LIN {X 0,Y 419.196,Z 864.185,A -85,B 0,C 180,E1 19901.419,E2 19901.419} C_VEL
LIN {X 0,Y 418.339,Z 869.705,A -85,B 0,C 180,E1 19898.661,E2 19898.661} C_VEL
LIN {X 0,Y 417.806,Z 873.843,A -85,B 0,C 180,E1 19895.769,E2 19895.769} C_VEL
LIN {X 0,Y 417.544,Z 876.277,A -85,B 0,C 180,E1 19893.02,E2 19893.02} C_VEL
LIN {X 0,Y 417.459,Z 877.198,A -85,B 0,C 180,E1 19890.137,E2 19890.137} C_VEL
LIN {X 0,Y 417.51,Z 876.519,A -85,B 0,C 180,E1 19887.392,E2 19887.392} C_VEL
LIN {X 0,Y 417.764,Z 874.258,A -85,B 0,C 180,E1 19884.506,E2 19884.506} C_VEL
LIN {X 0,Y 418.227,Z 870.613,A -85,B 0,C 180,E1 19881.753,E2 19881.753} C_VEL
LIN {X 0,Y 419.071,Z 865.05,A -85,B 0,C 180,E1 19878.857,E2 19878.857} C_VEL
LIN {X 0,Y 420.276,Z 858.016,A -85,B 0,C 180,E1 19876.094,E2 19876.094} C_VEL
LIN {X 0,Y 421.971,Z 849.236,A -85,B 0,C 180,E1 19873.339,E2 19873.339} C_VEL
LIN {X 0,Y 424.212,Z 838.486,A -85,B 0,C 180,E1 19870.589,E2 19870.589} C_VEL
LIN {X 0,Y 426.882,Z 826.191,A -85,B 0,C 180,E1 19867.99,E2 19867.99} C_VEL
LIN {X 0,Y 429.757,Z 813.215,A -85,B 0,C 180,E1 19865.681,E2 19865.681} C_VEL
LIN {X 0,Y 433.075,Z 797.976,A -85,B 0,C 180,E1 19863.39,E2 19863.39} C_VEL
LIN {X 0,Y 436.501,Z 781.676,A -85,B 0,C 180,E1 19861.323,E2 19861.323} C_VEL
LIN {X 0,Y 440.028,Z 763.676,A -85,B 0,C 180,E1 19859.403,E2 19859.403} C_VEL
LIN {X 0,Y 443.454,Z 744.549,A -85,B 0,C 180,E1 19857.698,E2 19857.698} C_VEL
LIN {X 0,Y 446.63,Z 724.241,A -85,B 0,C 180,E1 19856.198,E2 19856.198} C_VEL
LIN {X 0,Y 449.363,Z 703.738,A -85,B 0,C 180,E1 19854.965,E2 19854.965} C_VEL
LIN {X 0,Y 451.591,Z 682.841,A -85,B 0,C 180,E1 19853.956,E2 19853.956} C_VEL
LIN {X 0,Y 453.312,Z 661.563,A -85,B 0,C 180,E1 19853.163,E2 19853.163} C_VEL
LIN {X 0,Y 456.433,Z 619.357,A -85,B 0,C 180,E1 19851.962,E2 19851.962} C_VEL
LIN {X 0,Y 462.05,Z 551.52,A -85,B 0,C 180,E1 19850.353,E2 19850.353} C_VEL
LIN {X 0,Y 466.509,Z 485.901,A -85,B 0,C 180,E1 19849.025,E2 19849.025} C_VEL
LIN {X 0,Y 469.976,Z 414.611,A -85,B 0,C 180,E1 19847.825,E2 19847.825} C_VEL
LIN {X 0,Y 471.052,Z 393.311,A -85,B 0,C 180,E1 19847.463,E2 19847.463} C_VEL
LIN {X 0,Y 476.185,Z 369.743,A -85,B 0,C 180,E1 19846.561,E2 19846.561} C_VEL
LIN {X 0,Y 476.556,Z 345.293,A -85,B 0,C 180,E1 19844.828,E2 19844.828} C_VEL
LIN {X 0,Y 469.126,Z 324.998,A -85,B 0,C 180,E1 19842.175,E2 19842.175} C_VEL
LIN {X 0,Y 462.685,Z 309.482,A -85,B 0,C 180,E1 19839.929,E2 19839.929} C_VEL
LIN {X 0,Y 456.022,Z 295.191,A -85,B 0,C 180,E1 19837.67,E2 19837.67} C_VEL
LIN {X 0,Y 447.821,Z 279.246,A -85,B 0,C 180,E1 19834.862,E2 19834.862} C_VEL
LIN {X 0,Y 439.708,Z 265.393,A -85,B 0,C 180,E1 19832.149,E2 19832.149} C_VEL
LIN {X 0,Y 435.741,Z 259.224,A -85,B 0,C 180,E1 19830.778,E2 19830.778} C_VEL
LIN {X 0,Y 433.247,Z 255.233,A -85,B 0,C 180,E1 19829.901,E2 19829.901} C_VEL
LIN {X 0,Y 430.503,Z 250.807,A -85,B 0,C 180,E1 19828.888,E2 19828.888} C_VEL
LIN {X 0,Y 427.306,Z 246.461,A -85,B 0,C 180,E1 19827.753,E2 19827.753} C_VEL
LIN {X 0,Y 426.374,Z 244.715,A -85,B 0,C 180,E1 19827.364,E2 19827.364} C_VEL
LIN {X 0,Y 423.833,Z 241.89,A -85,B 0,C 180,E1 19826.48,E2 19826.48} C_VEL
LIN {X 0,Y 422.541,Z 239.071,A -85,B 0,C 180,E1 19825.887,E2 19825.887} C_VEL
LIN {X 0,Y 419.683,Z 236.312,A -85,B 0,C 180,E1 19824.867,E2 19824.867} C_VEL
LIN {X 0,Y 418.562,Z 233.254,A -85,B 0,C 180,E1 19824.261,E2 19824.261} C_VEL
LIN {X 0,Y 418.538,Z 233.089,A -85,B 0,C 180,E1 19820.53,E2 19820.53} C_VEL
LIN {X 0,Y 418.533,Z 233.058,A -85,B 0,C 180,E1 19816.66,E2 19816.66} C_VEL
LIN {X 0,Y 418.534,Z 233.043,A -85,B 0,C 180,E1 19812.837,E2 19812.837} C_VEL
LIN {X 0,Y 418.54,Z 233.095,A -85,B 0,C 180,E1 19808.933,E2 19808.933} C_VEL
LIN {X 0,Y 418.532,Z 233.045,A -85,B 0,C 180,E1 19805.071,E2 19805.071} C_VEL
LIN {X 0,Y 418.529,Z 233.064,A -85,B 0,C 180,E1 19801.232,E2 19801.232} C_VEL
LIN {X 0,Y 418.52,Z 233.07,A -85,B 0,C 180,E1 19797.398,E2 19797.398} C_VEL
LIN {X 0,Y 418.513,Z 233.043,A -85,B 0,C 180,E1 19793.553,E2 19793.553} C_VEL
LIN {X 0,Y 418.52,Z 233.1,A -85,B 0,C 180,E1 19789.678,E2 19789.678} C_VEL
LIN {X 0,Y 418.52,Z 233.096,A -85,B 0,C 180,E1 19785.754,E2 19785.754} C_VEL
LIN {X 0,Y 418.525,Z 233.086,A -85,B 0,C 180,E1 19781.906,E2 19781.906} C_VEL
LIN {X 0,Y 418.533,Z 233.168,A -85,B 0,C 180,E1 19781.072,E2 19781.072} C_VEL
LIN {X 0,Y 419.796,Z 236.493,A -85,B 0,C 180,E1 19780.376,E2 19780.376} C_VEL
LIN {X 0,Y 421.099,Z 238.531,A -85,B 0,C 180,E1 19779.861,E2 19779.861} C_VEL
LIN {X 0,Y 423.255,Z 242.427,A -85,B 0,C 180,E1 19778.956,E2 19778.956} C_VEL
LIN {X 0,Y 430.88,Z 257.106,A -85,B 0,C 180,E1 19775.748,E2 19775.748} C_VEL
LIN {X 0,Y 439.608,Z 273.969,A -85,B 0,C 180,E1 19772.354,E2 19772.354} C_VEL
LIN {X 0,Y 449.782,Z 294.439,A -85,B 0,C 180,E1 19768.655,E2 19768.655} C_VEL
LIN {X 0,Y 459.809,Z 315.283,A -85,B 0,C 180,E1 19765.268,E2 19765.268} C_VEL
LIN {X 0,Y 464.788,Z 325.491,A -85,B 0,C 180,E1 19763.767,E2 19763.767} C_VEL
LIN {X 0,Y 480.323,Z 350.017,A -85,B 0,C 180,E1 19761.525,E2 19761.525} C_VEL
LIN {X 0,Y 480.604,Z 356.269,A -85,B 0,C 180,E1 19761.342,E2 19761.342} C_VEL
